# B&R Automation Studio project Nitto (part 6)

#### l2str.ab
```automation-basic
(********************************************************************
 * COPYRIGHT -- Microsoft
 ********************************************************************
 * Library: HlpStr
 * File: l2str.ab
 * Author: beutert
 * Created: March 25, 2011
 ********************************************************************
 * Implementation of library HlpStr
 ********************************************************************
 Function: convert an UDINT value to string

    input:  value (UDINT)
						pointer to string (UDINT)
   output:  strlen (UINT)
 ********************************************************************)

FUNCTION l2str
	brsstrcpy(pString,"");

	lRest = value;

	if (value > 0) then
		loop ii=9 downto 0 do
			lDivisor = UDINT(brmpow(10,ii));
			lQuot = lRest / lDivisor;
			lRest = lRest MOD lDivisor;
			if (lRest <> value) then
				brsitoa(lQuot, adr(szQuot));
				brsstrcat(pString, adr(szQuot));
			endif
		endloop;
	else
		brsstrcpy(pString,"0");
	endif;

	l2str = UINT(brsstrlen(pString));

END_FUNCTION
```

#### RTRIM.ab
```automation-basic
(********************************************************************
 * COPYRIGHT -- Microsoft
 ********************************************************************
 * Library: HlpStr
 * File: RTRIM.ab
 * Author: beutert
 * Created: April 08, 2011
 ********************************************************************
 * Implementation of library HlpStr
 ********************************************************************
 Function: delete blanks at end of string

    input:  pointer to string (UDINT)
   output:  status
 ********************************************************************)

FUNCTION RTRIM
	if (enable = true) then
		wStrLenHlp = UINT(sizeof(szHlpStr1) - 1);
		wStrLen = UINT(brsstrlen(pString));
		if (wStrLen > wStrLenHlp) then
			status = 50000;	//string too long
		else
			status = 65535;
			brsstrcpy(adr(szHlpStr1),pString);
			loop
				pByte access adr(szHlpStr1)+ wStrLen-1;
				bDbg = pByte;	//nur für Monitor
				if (pByte = ' ') then
					szHlpStr1 = LEFT(szHlpStr1, INT(wStrLen) - 1);
					wStrLen = wStrLen - 1;
				else
					exitif (1=1);
				endif;
			endloop;
			brsstrcpy(pString,adr(szHlpStr1));
			status = 0;
		endif;
	else
		status = 65534;
	endif;
	RTRIM = status;
END_FUNCTION
```

#### TRIM.ab
```automation-basic
(********************************************************************
 * COPYRIGHT -- Microsoft
 ********************************************************************
 * Library: HlpStr
 * File: TRIM.ab
 * Author: beutert
 * Created: April 08, 2011
 ********************************************************************
 * Implementation of library HlpStr
 ********************************************************************
 Function: delete blanks at beginning and end of string

    input:  pointer to string (UDINT)
   output:  status
 ********************************************************************)

FUNCTION TRIM
	if (enable = true) then
		status = RTRIM(enable, pString);
		if (status = 0) then
			status = LTRIM(enable, pString);
		endif;
	else
		status = 65534;
	endif;
	TRIM = status;
END_FUNCTION
```

### Library Logical/Libraries/SwitchConf (IEC, version 1.01.0)
Depends on: Acp10man, Acp10_MC

#### SwitchConf.typ - Exported data types
```iecst
(********************************************************************
 * COPYRIGHT -- Bernecker + Rainer
 ********************************************************************
 * Library: SwitchConf
 * File: SwitchConf.typ
 * Author: hagera
 * Created: March 01, 2010
 ********************************************************************
 * Data types of library SwitchConf
 ********************************************************************)

TYPE
	StepDescription_typ :
		( (*STEP description typ*)
		WAIT := 0, (*wait for start command*)
		CHECK_INPUT_DATA, (*check input data for FB*)
		GET_OFFSET_POS_END_SWITCH, (*get offset for positive end switch*)
		GET_OFFSET_NEG_END_SWITCH, (*get offstet for negative end switch*)
		GET_OFFSET_REF_SWITCH, (*get offset for reference switch*)
		DEFINE_PARAMETER_LIST, (*define entries for parameter list*)
		WRITE_PARAMETER_LIST (*write parameter list to axis*)
		);
	SwitchConfiguration_typ : 	STRUCT  (*single switch configuration typ*)
		ioInformation : PLACTION_GET_CROSSLINK_INFO_typ; (*i/o information for switch*)
		Status : UINT; (*status of i/o information*)
		Offset : UINT; (*offset of i/o in data*)
		shiftBits : UINT; (*bits to shift*)
	END_STRUCT;
	SwitchesACPm_typ : 	STRUCT  (*switches for ACPm typ*)
		posEndSwitch : SwitchConfiguration_typ; (*positive end switch*)
		negEndSwitch : SwitchConfiguration_typ; (*negative end switch*)
		refSwitch : SwitchConfiguration_typ; (*reference switch*)
	END_STRUCT;
	ErrorNumbers_typ :
		(
		OK := 0, (*no error*)
		INVALID_AXIS_REFERENCE := 50001, (*error number for invalid axis reference*)
		INVALID_DEVICE_NAME, (*error number for invalid device name*)
		INVALID_CHANNEL_NAME, (*error number for invalid channel name*)
		ERROR_GET_OFFSET_FOR_SWITCH, (*error number for getting offset for switch*)
		ERROR_WRITE_PARAMETER_LIST (*error number for writing parameter list*)
		);
	ParameterList_typ : 	STRUCT  (*parameter list typ*)
		List : ARRAY[0..30] OF ACP10PRB06_typ; (*parameter list*)
		listInfo : ACP10DATBL_typ; (*parameter list info*)
		configMaCyclicPos : ARRAY[0..1] OF UINT; (*MaCyclicPos*)
		ui2 : UINT; (*value data type UINT*)
		ui4 : UDINT; (*value data type UDINT*)
		Execute : BOOL; (*execute parameter list write*)
		Counter : USINT; (*parameter counter*)
	END_STRUCT;
END_TYPE
```

#### SwitchConf.fun - Exported functions and function blocks
```iecst
(********************************************************************
 * COPYRIGHT -- Bernecker + Rainer
 ********************************************************************
 * Library: SwitchConf
 * File: SwitchConf.fun
 * Author: hagera
 * Created: March 01, 2010
 ********************************************************************
 * Functions and function blocks of library SwitchConf
 ********************************************************************)

FUNCTION_BLOCK SwitchConfiguration (*FUB to configure end-switches and ref-switch for AcoposMulti*)
	VAR_INPUT
		Axis : UDINT; (*axis reference*)
		Execute : BOOL; (*start initialization at rising edge*)
		posEndSwitchDeviceName : UDINT; (*device name of module where positive end switch is connected*)
		posEndSwitchChannelName : UDINT; (*channel name of i/o where positive end switch is connected*)
		negEndSwitchDeviceName : UDINT; (*device name of module where negative end switch is connected*)
		negEndSwitchChannelName : UDINT; (*channel name of i/o where negative end switch is connected*)
		refSwitchDeviceName : UDINT; (*device name of module where reference switch is connected*)
		refSwitchChannelName : UDINT; (*channel name of i/o where reference switch is connected*)
	END_VAR
	VAR_OUTPUT
		Done : BOOL; (*initialization complete*)
		Busy : BOOL; (*initialization active*)
		Error : BOOL; (*error occured in FB*)
		ErrorID : ErrorNumbers_typ; (*error number*)
		ErrorInitparalist :UINT;
	END_VAR
	VAR
		zzEdge00000 :BOOL;
		Step : StepDescription_typ; (*intern variable*)
		Switches : SwitchesACPm_typ; (*intern variable*)
		Parameter : ParameterList_typ; (*intern variable*)
		MC_BR_InitParList_Switch : MC_BR_InitParList; (*intern variable*)
	END_VAR
END_FUNCTION_BLOCK
```

#### SwitchConfiguration.st - FUB to configure end-switches and ref-switch for ACOPOSmulti
```iecst
(********************************************************************
 * COPYRIGHT -- Bernecker + Rainer
 ********************************************************************
 * Library: SwitchConf
 * File: SwitchConfiguration.st
 * Author: hagera
 * Created: March 01, 2010
 ********************************************************************
 * Implementation of library SwitchConf
 *
 * History:
 * 2012-07-25 /schoenefeldr/
 * 		Change IPL-mode of ACP10PAR_MAx_CYCLIC_POS only if it is used
 *
 *
 *
 *
 ********************************************************************)

(* FUB to configure end-switches and ref-switch for ACOPOSmulti *)
FUNCTION_BLOCK SwitchConfiguration

CASE Step OF
	WAIT:
		IF (EDGEPOS(Execute) = 1) THEN
			Done := 0;
			Busy := 1;
			Error := 0;
			ErrorID := 0;
			Step := CHECK_INPUT_DATA;
		END_IF

	CHECK_INPUT_DATA :
		IF (Axis = 0) THEN
			Busy := 0;
			Error := 1;
			ErrorID := INVALID_AXIS_REFERENCE;
			Step := WAIT;
		ELSIF (posEndSwitchDeviceName = 0 AND negEndSwitchDeviceName = 0 AND refSwitchDeviceName = 0) OR
			(posEndSwitchDeviceName = 0 AND posEndSwitchChannelName <> 0) OR
   			(negEndSwitchDeviceName = 0 AND negEndSwitchChannelName <> 0) OR
   			(refSwitchDeviceName = 0 AND refSwitchChannelName <> 0)	THEN
			Busy := 0;
			Error := 1;
			ErrorID := INVALID_DEVICE_NAME;
			Step := WAIT;
		ELSIF (posEndSwitchDeviceName <> 0 AND posEndSwitchChannelName = 0) OR
			(negEndSwitchDeviceName <> 0 AND negEndSwitchChannelName = 0) OR
			(refSwitchDeviceName <> 0 AND refSwitchChannelName = 0) THEN
   			Busy := 0;
			Error := 1;
			ErrorID := INVALID_CHANNEL_NAME;
			Step := WAIT;
		ELSE
			Step := GET_OFFSET_POS_END_SWITCH;
		END_IF

	GET_OFFSET_POS_END_SWITCH :
		IF (posEndSwitchDeviceName = 0) THEN
			Step := GET_OFFSET_NEG_END_SWITCH;
		ELSE
			Switches.posEndSwitch.ioInformation.DeviceName := posEndSwitchDeviceName;
			Switches.posEndSwitch.ioInformation.ChannelName := posEndSwitchChannelName;

			Switches.posEndSwitch.Status := plAction(0, plACTION_GET_CROSSLINK_INFO, ADR(Switches.posEndSwitch.ioInformation), SIZEOF(Switches.posEndSwitch.ioInformation));

			IF (Switches.posEndSwitch.Status = 0) THEN
				Switches.posEndSwitch.Offset := (Switches.posEndSwitch.ioInformation.Offset / 32) * 32;
				Switches.posEndSwitch.shiftBits := Switches.posEndSwitch.ioInformation.Offset MOD 32;
				Step := GET_OFFSET_NEG_END_SWITCH;
			ELSE
				Busy := 0;
				Error := 1;
				ErrorID := ERROR_GET_OFFSET_FOR_SWITCH;
				Step := WAIT;
   			END_IF
		END_IF

	GET_OFFSET_NEG_END_SWITCH :
		IF (negEndSwitchDeviceName = 0) THEN
			Step := GET_OFFSET_REF_SWITCH;
		ELSE
			Switches.negEndSwitch.ioInformation.DeviceName := negEndSwitchDeviceName;
			Switches.negEndSwitch.ioInformation.ChannelName := negEndSwitchChannelName;

			Switches.negEndSwitch.Status := plAction(0, plACTION_GET_CROSSLINK_INFO, ADR(Switches.negEndSwitch.ioInformation), SIZEOF(Switches.negEndSwitch.ioInformation));

			IF (Switches.negEndSwitch.Status = 0) THEN
				Switches.negEndSwitch.Offset := (Switches.negEndSwitch.ioInformation.Offset / 32) * 32;
				Switches.negEndSwitch.shiftBits := Switches.negEndSwitch.ioInformation.Offset MOD 32;
				Step := GET_OFFSET_REF_SWITCH;
			ELSE
				Busy := 0;
				Error := 1;
				ErrorID := ERROR_GET_OFFSET_FOR_SWITCH;
				Step := WAIT;
   			END_IF
		END_IF

	GET_OFFSET_REF_SWITCH  :
		IF (refSwitchDeviceName = 0) THEN
			Step := DEFINE_PARAMETER_LIST;
		ELSE
			Switches.refSwitch.ioInformation.DeviceName := refSwitchDeviceName;
			Switches.refSwitch.ioInformation.ChannelName := refSwitchChannelName;

			Switches.refSwitch.Status := plAction(0, plACTION_GET_CROSSLINK_INFO, ADR(Switches.refSwitch.ioInformation), SIZEOF(Switches.refSwitch.ioInformation));

			IF (Switches.refSwitch.Status = 0) THEN
				Switches.refSwitch.Offset := (Switches.refSwitch.ioInformation.Offset / 32) * 32;
				Switches.refSwitch.shiftBits := Switches.refSwitch.ioInformation.Offset MOD 32;
				Step := DEFINE_PARAMETER_LIST;
			ELSE
				Busy := 0;
				Error := 1;
				ErrorID := ERROR_GET_OFFSET_FOR_SWITCH;
				Step := WAIT;
   			END_IF
		END_IF

	DEFINE_PARAMETER_LIST :
		Parameter.List[0].par_id := ACP10PAR_FUNCTION_BLOCK_CREATE;
		Parameter.ui2 := ACP10PAR_BIT_MODE;
		memcpy(ADR(Parameter.List[0].data_byte[0]), ADR(Parameter.ui2), SIZEOF(Parameter.ui2));
		Parameter.Counter := Parameter.Counter + 1;

		Parameter.List[Parameter.Counter].par_id := ACP10PAR_BIT_A1;
		Parameter.ui4 := 1;
		memcpy(ADR(Parameter.List[Parameter.Counter].data_byte[0]), ADR(Parameter.ui4), SIZEOF(Parameter.ui4));
		Parameter.Counter := Parameter.Counter + 1;

		Parameter.List[Parameter.Counter].par_id := ACP10PAR_BIT_A2;
		Parameter.ui4 := 1;
		memcpy(ADR(Parameter.List[Parameter.Counter].data_byte[0]), ADR(Parameter.ui4), SIZEOF(Parameter.ui4));
		Parameter.Counter := Parameter.Counter + 1;

		Parameter.List[Parameter.Counter].par_id := ACP10PAR_BIT_A3;
		Parameter.ui4 := 1;
		memcpy(ADR(Parameter.List[Parameter.Counter].data_byte[0]), ADR(Parameter.ui4), SIZEOF(Parameter.ui4));
		Parameter.Counter := Parameter.Counter + 1;

		Parameter.List[Parameter.Counter].par_id := ACP10PAR_BIT_IN1_PARID;
		Parameter.ui2 := ACP10PAR_MA1_CYCLIC_POS;
		memcpy(ADR(Parameter.List[Parameter.Counter].data_byte[0]), ADR(Parameter.ui2), SIZEOF(Parameter.ui2));
		Parameter.Counter := Parameter.Counter + 1;

		Parameter.List[Parameter.Counter].par_id := ACP10PAR_BIT_IN2_PARID;
		Parameter.ui2 := ACP10PAR_MA2_CYCLIC_POS;
		memcpy(ADR(Parameter.List[Parameter.Counter].data_byte[0]), ADR(Parameter.ui2), SIZEOF(Parameter.ui2));
		Parameter.Counter := Parameter.Counter + 1;

		Parameter.List[Parameter.Counter].par_id := ACP10PAR_BIT_IN3_PARID;
		Parameter.ui2 := ACP10PAR_MA3_CYCLIC_POS;
		memcpy(ADR(Parameter.List[Parameter.Counter].data_byte[0]), ADR(Parameter.ui2), SIZEOF(Parameter.ui2));
		Parameter.Counter := Parameter.Counter + 1;

		Parameter.List[Parameter.Counter].par_id := ACP10PAR_BIT_MODE;
		Parameter.ui2 := 10;
		memcpy(ADR(Parameter.List[Parameter.Counter].data_byte[0]), ADR(Parameter.ui2), SIZEOF(Parameter.ui2));
		Parameter.Counter := Parameter.Counter + 1;

		IF (posEndSwitchDeviceName <> 0) THEN
			// 2012-07-25 /schoenefeldr/
			// Moved here into configuration dependent section
			Parameter.List[Parameter.Counter].par_id := ACP10PAR_MA1_CYCLIC_IPL_MODE;
			Parameter.List[Parameter.Counter].data_byte[0] := 0;
			Parameter.Counter := Parameter.Counter + 1;

			Parameter.List[Parameter.Counter].par_id := ACP10PAR_CYCLIC_DP_DATA_OFFSET;
			Parameter.ui2 := Switches.posEndSwitch.Offset;
			memcpy(ADR(Parameter.List[Parameter.Counter].data_byte[0]), ADR(Parameter.ui2), SIZEOF(Parameter.ui2));
			Parameter.Counter := Parameter.Counter + 1;

			Parameter.List[Parameter.Counter].par_id := ACP10PAR_CYCLIC_DP_DATA_TYPE;
			Parameter.ui2 := 7;
			memcpy(ADR(Parameter.List[Parameter.Counter].data_byte[0]), ADR(Parameter.ui2), SIZEOF(Parameter.ui2));
			Parameter.Counter := Parameter.Counter + 1;

			Parameter.configMaCyclicPos[0] := Switches.posEndSwitch.ioInformation.NodeId;
			Parameter.configMaCyclicPos[1] := ACP10PAR_CYCLIC_DP_DATA_OFFSET;

			Parameter.List[Parameter.Counter].par_id := ACP10PAR_CONFIG_MA1_CYCLIC_POS;
			memcpy(ADR(Parameter.List[Parameter.Counter].data_byte[0]), ADR(Parameter.configMaCyclicPos), SIZEOF(Parameter.configMaCyclicPos));
			Parameter.Counter := Parameter.Counter + 1;

			Parameter.List[Parameter.Counter].par_id := ACP10PAR_BIT_B1+0;
			Parameter.ui4 := Switches.posEndSwitch.shiftBits;
			memcpy(ADR(Parameter.List[Parameter.Counter].data_byte[0]), ADR(Parameter.ui4), SIZEOF(Parameter.ui4));
			Parameter.Counter := Parameter.Counter + 1;

			Parameter.List[Parameter.Counter].par_id := ACP10PAR_POS_LIMIT_SWITCH_PARID;
			Parameter.ui2 := ACP10PAR_BIT_VALUE1;
			memcpy(ADR(Parameter.List[Parameter.Counter].data_byte[0]), ADR(Parameter.ui2), SIZEOF(Parameter.ui2));
			Parameter.Counter := Parameter.Counter + 1;
		END_IF

		IF (negEndSwitchDeviceName <> 0) THEN
			// 2012-07-25 /schoenefeldr/
			// Moved here into configuration dependent section
			Parameter.List[Parameter.Counter].par_id := ACP10PAR_MA2_CYCLIC_IPL_MODE;
			Parameter.List[Parameter.Counter].data_byte[0] := 0;
			Parameter.Counter := Parameter.Counter + 1;

			Parameter.List[Parameter.Counter].par_id := ACP10PAR_CYCLIC_DP_DATA_OFFSET;
			Parameter.ui2 := Switches.negEndSwitch.Offset;
			memcpy(ADR(Parameter.List[Parameter.Counter].data_byte[0]), ADR(Parameter.ui2), SIZEOF(Parameter.ui2));
			Parameter.Counter := Parameter.Counter + 1;

			Parameter.List[Parameter.Counter].par_id := ACP10PAR_CYCLIC_DP_DATA_TYPE;
			Parameter.ui2 := 7;
			memcpy(ADR(Parameter.List[Parameter.Counter].data_byte[0]), ADR(Parameter.ui2), SIZEOF(Parameter.ui2));
			Parameter.Counter := Parameter.Counter + 1;

			Parameter.configMaCyclicPos[0] := Switches.negEndSwitch.ioInformation.NodeId;
			Parameter.configMaCyclicPos[1] := ACP10PAR_CYCLIC_DP_DATA_OFFSET;

			Parameter.List[Parameter.Counter].par_id := ACP10PAR_CONFIG_MA2_CYCLIC_POS;
			memcpy(ADR(Parameter.List[Parameter.Counter].data_byte[0]), ADR(Parameter.configMaCyclicPos), SIZEOF(Parameter.configMaCyclicPos));
			Parameter.Counter := Parameter.Counter + 1;

			Parameter.List[Parameter.Counter].par_id := ACP10PAR_BIT_B2+0;
			Parameter.ui4 := Switches.negEndSwitch.shiftBits;
			memcpy(ADR(Parameter.List[Parameter.Counter].data_byte[0]), ADR(Parameter.ui4), SIZEOF(Parameter.ui4));
			Parameter.Counter := Parameter.Counter + 1;

			Parameter.List[Parameter.Counter].par_id := ACP10PAR_NEG_LIMIT_SWITCH_PARID;
			Parameter.ui2 := ACP10PAR_BIT_VALUE2;
			memcpy(ADR(Parameter.List[Parameter.Counter].data_byte[0]), ADR(Parameter.ui2), SIZEOF(Parameter.ui2));
			Parameter.Counter := Parameter.Counter + 1;
		END_IF

		IF (refSwitchDeviceName <> 0) THEN
			// 2012-07-25 /schoenefeldr/
			// Moved here into configuration dependent section
			Parameter.List[Parameter.Counter].par_id := ACP10PAR_MA3_CYCLIC_IPL_MODE;
			Parameter.List[Parameter.Counter].data_byte[0] := 0;
			Parameter.Counter := Parameter.Counter + 1;

			Parameter.List[Parameter.Counter].par_id := ACP10PAR_CYCLIC_DP_DATA_OFFSET;
			Parameter.ui2 := Switches.refSwitch.Offset;
			memcpy(ADR(Parameter.List[Parameter.Counter].data_byte[0]), ADR(Parameter.ui2), SIZEOF(Parameter.ui2));
			Parameter.Counter := Parameter.Counter + 1;

			Parameter.List[Parameter.Counter].par_id := ACP10PAR_CYCLIC_DP_DATA_TYPE;
			Parameter.ui2 := 7;
			memcpy(ADR(Parameter.List[Parameter.Counter].data_byte[0]), ADR(Parameter.ui2), SIZEOF(Parameter.ui2));
			Parameter.Counter := Parameter.Counter + 1;

			Parameter.configMaCyclicPos[0] := Switches.refSwitch.ioInformation.NodeId;
			Parameter.configMaCyclicPos[1] := ACP10PAR_CYCLIC_DP_DATA_OFFSET;

			Parameter.List[Parameter.Counter].par_id := ACP10PAR_CONFIG_MA3_CYCLIC_POS;
			memcpy(ADR(Parameter.List[Parameter.Counter].data_byte[0]), ADR(Parameter.configMaCyclicPos), SIZEOF(Parameter.configMaCyclicPos));
			Parameter.Counter := Parameter.Counter + 1;

			Parameter.List[Parameter.Counter].par_id := ACP10PAR_BIT_B3+0;
			Parameter.ui4 := Switches.refSwitch.shiftBits;
			memcpy(ADR(Parameter.List[Parameter.Counter].data_byte[0]), ADR(Parameter.ui4), SIZEOF(Parameter.ui4));
			Parameter.Counter := Parameter.Counter + 1;

			Parameter.List[Parameter.Counter].par_id := ACP10PAR_REFERENCE_SWITCH_PARID;
			Parameter.ui2 := ACP10PAR_BIT_VALUE3;
			memcpy(ADR(Parameter.List[Parameter.Counter].data_byte[0]), ADR(Parameter.ui2), SIZEOF(Parameter.ui2));
			Parameter.Counter := Parameter.Counter + 1;
		END_IF

		Step := WRITE_PARAMETER_LIST;

	WRITE_PARAMETER_LIST :
		Parameter.listInfo.parameter.data_adr := ADR(Parameter.List);
		Parameter.listInfo.parameter.format := ncFORMAT_B06;
		Parameter.listInfo.parameter.data_len := Parameter.Counter * SIZEOF(ACP10PRB06_typ);
		Parameter.Execute := 1;

		IF (MC_BR_InitParList_Switch.Done = 1) THEN
			Parameter.Execute := 0;
			Busy := 0;
			Done := 1;
			Step := WAIT;
		ELSIF (MC_BR_InitParList_Switch.Error = 1) THEN
			Parameter.Execute := 0;
			Busy := 0;
			ErrorInitparalist := MC_BR_InitParList_Switch.ErrorID;
			Error := 1;
			ErrorID := ERROR_WRITE_PARAMETER_LIST;
			Step := WAIT;
		END_IF

		MC_BR_InitParList_Switch(Axis := Axis, Execute := Parameter.Execute, DataAddress := ADR(Parameter.listInfo));

END_CASE

END_FUNCTION_BLOCK
```

### Library Logical/Libraries/TorqueCtrl (IEC) - Torque control
Depends on: LoopConR, Acp10_MC

#### TorqueCtrl.typ - Exported data types
```iecst
(********************************************************************
 * COPYRIGHT -- Bernecker + Rainer
 ********************************************************************
 * Library: TorqueCtrl
 * File: TorqueCtrl.typ
 * Author: knausenbergl
 * Created: October 29, 2012
 ********************************************************************
 * Data types of library TorqueCtrl
 ********************************************************************)

TYPE
	TC_WINDER_IS_TYP : 	STRUCT
		RefTension : ARRAY[0..1]OF REAL;
		RefDiameter : ARRAY[0..1]OF REAL;
		SetLineSpeed : REAL;
		ActDiameter : REAL;
		SetWndSpeed : REAL;
		SetMotorTorque : REAL;
		LineUnits : REAL;
		LCRLimScal_Tension : LCRLimScal; (*scale tension force depending on actual diameter*)
		GearRatio : REAL;
		EncoderIf : ACP10ENCPA_typ;
		WndUnitsPerLoadRev : REAL; (*winder units per load revolution [Slave Units]*)
		SetTorqueRaw : REAL; (*raw, unlimited set torque [Nm]*)
		SetTension : REAL;
	END_STRUCT;
END_TYPE
```

#### TorqueCtrl.fun - Exported functions and function blocks
```iecst
(********************************************************************
 * COPYRIGHT -- Bernecker + Rainer
 ********************************************************************
 * Library: TorqueCtrl
 * File: TorqueCtrl.fun
 * Author: knausenbergl
 * Created: October 29, 2012
 ********************************************************************
 * Functions and function blocks of library TorqueCtrl
 ********************************************************************)

FUNCTION_BLOCK TC_Winder
	VAR_INPUT
		RefTension : ARRAY[0..1] OF REAL; (*reference material tension [N]*)
		RefDiameter : ARRAY[0..1] OF REAL; (*reference diameters corresponding to RefTension [Master Units]*)
		SetLineSpeed : REAL; (*line speed [Master Units / s]*)
		ActDiameter : REAL; (*actual winder diameter [Master Units]*)
		EncoderIf : ACP10ENCPA_typ; (*winder encoder interface*)
		GearRatio : REAL; (*motor rev. / winder rev. []*)
		LineUnits : REAL; (*line position scaling [Master Units / m]*)
	END_VAR
	VAR_OUTPUT
		SetWndSpeed : REAL; (*set winder speed [Slave Units / s]*)
		SetMotorTorque : REAL; (*set motor torque [Nm]*)
		SetTension : REAL; (*set material tension [N]*)
	END_VAR
	VAR
		IS : TC_WINDER_IS_TYP; (*internal data*)
	END_VAR
END_FUNCTION_BLOCK
```

#### TC_Winder.st
```iecst
(********************************************************************
 * COPYRIGHT -- Bernecker + Rainer
 ********************************************************************
 * Library: TorqueCtrl
 * File: TC_Winder.st
 * Author: knausenbergl
 * Created: October 29, 2012
 ********************************************************************
 * Implementation of library TorqueCtrl
 *
 * History:
 * 2012-10-29 /knausenbergl/
 *		Task created
 * 2012-10-31 /schoenefeldr/
 *		Removed unused dynamic adaptation of force
 * 2012-11-01 /schoenefeldr/
 *		Removed unused inputs
 ********************************************************************)

(* Calculate velocity and torque depending on force setpoint and diameter *)
FUNCTION_BLOCK TC_Winder

	//UPDATE FUB INPUTS
	IS.RefTension		:= RefTension;
	IS.RefDiameter		:= RefDiameter;
	IS.SetLineSpeed		:= SetLineSpeed;
	IS.ActDiameter		:= ActDiameter;
	IS.EncoderIf		:= EncoderIf;
	IS.GearRatio		:= GearRatio;
	IS.LineUnits		:= LineUnits;

	IS.WndUnitsPerLoadRev	:= UDINT_TO_REAL(IS.EncoderIf.scaling.load.units) * IS.GearRatio / UDINT_TO_REAL(IS.EncoderIf.scaling.load.rev_motor);

	//calculate set winder speed
	IF (IS.ActDiameter > 0.0) THEN
		IS.SetWndSpeed	:= IS.SetLineSpeed / (MATH_PI * IS.ActDiameter) * IS.WndUnitsPerLoadRev;
	ELSE
		IS.SetWndSpeed	:= 0.0;
	END_IF;

	//calculate set tension depending on actual diameter
	IS.LCRLimScal_Tension.x		:= IS.ActDiameter;
	IS.LCRLimScal_Tension.x1	:= IS.RefDiameter[0];
	IS.LCRLimScal_Tension.y1	:= IS.RefTension[0];
	IS.LCRLimScal_Tension.x2	:= IS.RefDiameter[1];
	IS.LCRLimScal_Tension.y2	:= IS.RefTension[1];
	IS.LCRLimScal_Tension();
	IS.SetTension	:= IS.LCRLimScal_Tension.y;
	IS.SetTorqueRaw	:= IS.LCRLimScal_Tension.y * IS.ActDiameter / (2.0 * IS.GearRatio * IS.LineUnits);

	//UPDATE FUB OUTPUTS
	SetWndSpeed		:= IS.SetWndSpeed;
	SetMotorTorque	:= IS.SetTorqueRaw;
	SetTension		:= IS.SetTension;

END_FUNCTION_BLOCK
```

### Library Logical/Libraries/UserVC (IEC, version 3.00.0)
Depends on: AsString, runtime

#### UserVC.var
```iecst
VAR CONSTANT
	ENABLE_NOT_SET	:UINT	:=65000;
	HEX_BASE	:SINT	:=16;
	SORTING_ABORTED	:UINT	:=6000;
	SORTING_BUSY	:UINT	:=65535;
	SORTING_NO_ERROR	:UINT	:=0;
	SORT_ALPHANUMERICALLY	:USINT	:=4;
	SORT_CASE_SENSITIVE1	:USINT	:=2;
	SORT_CASE_SENSITIVE2	:USINT	:=3;
	SWAP_FILENAMES	:USINT	:=1;
END_VAR
```

#### UserVC.fun
```iecst
FUNCTION_BLOCK Sort
	VAR_INPUT
		enable : BOOL;
		pStringArray : UDINT;
		StringLen : UINT;
		ArrayLen : UINT;
	END_VAR
	VAR_OUTPUT
		Status : UINT;
	END_VAR
	VAR
		xcnt : UINT;
		ycnt : UINT;
		StepCounter : UINT;
		SortStep : USINT;
		FileNameBuffer : STRING[80];
		pChar1 : REFERENCE TO USINT;
		pChar2 : REFERENCE TO USINT;
	END_VAR
END_FUNCTION_BLOCK

FUNCTION_BLOCK ConvertHex
	VAR_INPUT
		Enable : BOOL;
		pHexValue : UDINT;
		DecValue : UDINT;
		SizeDecValue : USINT;
	END_VAR
	VAR_OUTPUT
		Status : UINT;
	END_VAR
	VAR
		HexASCII : ARRAY[0..7] OF USINT;
		Index : SINT;
		End : USINT;
		Rest : UDINT;
	END_VAR
END_FUNCTION_BLOCK
```

#### Sort.st
```iecst
FUNCTION_BLOCK Sort
(* Implementation of sort *)

(**********************************************************************************************************************)
(* Object name: sort                                                                                                                              	*)
(* Author:      Peter Hauser,  B&R                                                                                                               	*)
(* Site:        Eggelsberg                                                                                                                             	*)
(* Created:     25-aug-2003                                                                                                                           	*)
(* Restriction: ------                                                                                                                          	*)
(* Description: The Sort-Function sorts a String Array alphanumerically                                                                                                                                       	*)
(*                                                                                                                                                              	*)
(*----------------------------------------------------------------------------------------------------------------------------------------	*)
(* Version 1.00.1   25-aug-2003  Peter Hauser									*)
(*----------------------------------------------------------------------------------------------------------------------------------------	*)
(* Development tool: B&R Automation Studio V2.3.0.9 							*)
(*----------------------------------------------------------------------------------------------------------------------------------------	*)
(* Comment:                                                                                                                     			*)
(**********************************************************************************************************************)

(* Errors *)

IF ((enable = 0) AND (StepCounter > 0) AND (StepCounter < ((ArrayLen / StringLen) - 1))) THEN
	Status:= SORTING_ABORTED;

ELSIF ((enable = 1) AND (StepCounter >= 0) AND (StepCounter < ((ArrayLen / StringLen) - 1))) THEN
	Status:= SORTING_BUSY;

ELSE
	Status:= SORTING_NO_ERROR;

END_IF

(* sorting StringArray alphanumerically *)

IF ((enable = 1) AND ((Status = 0) OR (Status = 65535))) THEN

	FOR xcnt:= 0 TO ((ArrayLen / StringLen) - 2) DO

		FOR ycnt:= 0 TO StringLen DO
			(* read characters of FileNames *)
			pChar1 ACCESS (pStringArray + (StringLen * xcnt) + ycnt);
			pChar2 ACCESS (pStringArray + (StringLen * xcnt) + StringLen + ycnt);

			(* if no data in FileName1 -> Swap FileNames *)
			IF ((ycnt = 0) AND (pChar1 = 0) AND (pChar2 > 0)) THEN
				SortStep:= SWAP_FILENAMES;

			(* if no data in FileName2 -> next 2 FileNames *)
			ELSIF ((ycnt = 0) AND (pChar2 = 0)) THEN
				EXIT;

			(* if data in both FileNames *)
			ELSE
				(* detect case of letters *)
				IF ((pChar1 >= 65) AND (pChar1 <= 90) AND (pChar2 >= 97) AND (pChar2 <= 122)) THEN
					SortStep:= SORT_CASE_SENSITIVE1;

				ELSIF ((pChar1 >= 97) AND (pChar1 <= 122) AND (pChar2 >= 65) AND (pChar2 <= 90)) THEN
					SortStep:= SORT_CASE_SENSITIVE2;

				(* if characters are equal -> compare next characters of FileName *)
				ELSIF ((pChar1 = pChar2) AND (pChar2 <> 0)) THEN
					SortStep:= 0;

				(* if both FileNames are finished *)
				ELSIF ((pChar1 = 0) AND (pChar2 = 0)) THEN
					EXIT;

				(* sort Alphanumerically *)
				ELSE
					SortStep:= SORT_ALPHANUMERICALLY;
				END_IF
			END_IF

			CASE SortStep OF

				SWAP_FILENAMES:
					memcpy(ADR(FileNameBuffer), (pStringArray + (StringLen * xcnt)), StringLen);
					memcpy((pStringArray + (StringLen * xcnt)), (pStringArray + (StringLen * xcnt) + StringLen), StringLen);
					memcpy((pStringArray + (StringLen * xcnt) + StringLen), ADR(FileNameBuffer), StringLen);
					EXIT;

				SORT_CASE_SENSITIVE1:
					IF (pChar2 <= (pChar1 + 32)) THEN
						memcpy(ADR(FileNameBuffer), (pStringArray + (StringLen * xcnt)), StringLen);
						memcpy((pStringArray + (StringLen * xcnt)), (pStringArray + (StringLen * xcnt) + StringLen), StringLen);
						memcpy((pStringArray + (StringLen * xcnt) + StringLen), ADR(FileNameBuffer), StringLen);
						EXIT;
					ELSE
						EXIT;
					END_IF

				SORT_CASE_SENSITIVE2:
					IF (pChar2 < (pChar1 - 32)) THEN
						memcpy(ADR(FileNameBuffer), (pStringArray + (StringLen * xcnt)), StringLen);
						memcpy((pStringArray + (StringLen * xcnt)), (pStringArray + (StringLen * xcnt) + StringLen), StringLen);
						memcpy((pStringArray + (StringLen * xcnt) + StringLen), ADR(FileNameBuffer), StringLen);
						EXIT;
					ELSE
						EXIT;
					END_IF

				SORT_ALPHANUMERICALLY:
					IF pChar1 > pChar2 THEN
						memcpy(ADR(FileNameBuffer), (pStringArray + (StringLen * xcnt)), StringLen);
						memcpy((pStringArray + (StringLen * xcnt)), (pStringArray + (StringLen * xcnt) + StringLen), StringLen);
						memcpy((pStringArray + (StringLen * xcnt) + StringLen), ADR(FileNameBuffer), StringLen);
						EXIT;
					ELSE
						EXIT;
					END_IF

			END_CASE
		END_FOR

	END_FOR

	(* execute sorting [NumStringsToSort] times *)
	IF xcnt = ((ArrayLen / StringLen) - 1) THEN
		StepCounter:= StepCounter + 1;
	END_IF;

	IF StepCounter >= (ArrayLen / StringLen) THEN
		StepCounter:= 0;
	END_IF

END_IF			(* if enable = 1 *)

END_FUNCTION_BLOCK
```

#### ConvertHex.st
```iecst
FUNCTION_BLOCK ConvertHex
(* Implementation of ConvertHex *)

(**********************************************************************************************************************)
(* Object name: ConvertHex                                                                                                                              	*)
(* Author:      Christoph Trappl,  B&R                                                                                                               	*)
(* Site:        Eggelsberg                                                                                                                             	*)
(* Created:     27-aug-2003                                                                                                                           	*)
(* Restriction: -----                                                                                                                          	*)
(* Description: Converts a decimal value to hexadecimal ASCII                                                                                                                                	*)
(*                                                                                                                                                              	*)
(*----------------------------------------------------------------------------------------------------------------------------------------	*)
(* Version 1.00.1   27-aug-2003  Christoph Trappl								*)
(*----------------------------------------------------------------------------------------------------------------------------------------	*)
(* Version 1.00.2   02-feb-2004  Peter Hauser									*)
(*----------------------------------------------------------------------------------------------------------------------------------------	*)
(* Development tool: B&R Automation Studio V2.3.0.9 							*)
(*----------------------------------------------------------------------------------------------------------------------------------------	*)
(* Comment:                                                                                                                     			*)
(**********************************************************************************************************************)

(* Execute Functionblock when enable = true *)
IF (Enable = 1) THEN

//210812,TB: CONSTANT EXECUTION_BUSY replaced	by standard
//	Status := EXECUTION_BUSY;
	Status := ERR_FUB_BUSY;

	(* reset the complete memory area, that will be overwritten during the function execution *)
	memset(pHexValue, 0, SIZEOF(HexASCII));

	HexASCII[0]:= 0;
	HexASCII[1]:= 0;
	HexASCII[2]:= 0;
	HexASCII[3]:= 0;
	HexASCII[4]:= 0;
	HexASCII[5]:= 0;
	HexASCII[6]:= 0;
	HexASCII[7]:= 0;

	IF SizeDecValue = 0 THEN
		IF (DecValue > 16#FFFFFFF)  THEN
			Index:= 7;
		ELSIF (DecValue > 16#FFFFFF) THEN
			Index:= 6;
		ELSIF (DecValue > 16#FFFFF) THEN
			Index:= 5;
		ELSIF (DecValue > 16#FFFF) THEN
			Index:= 4;
		ELSIF (DecValue > 16#FFF) THEN
			Index:= 3;
		ELSIF (DecValue > 16#FF) THEN
			Index:= 2;
		ELSIF (DecValue > 16#F) THEN
			Index:= 1;
		ELSE
			Index:= 0;
		END_IF
	ELSIF SizeDecValue = 1 THEN
		Index:= 1;
	ELSIF SizeDecValue = 2 THEN
		Index:= 3;
	ELSIF SizeDecValue = 4 THEN
		Index:= 7;
	END_IF

	REPEAT
		IF DecValue > 0 OR SizeDecValue > 0 THEN
			End:= 0;
			Rest:= DecValue MOD HEX_BASE;
			DecValue:= DecValue / HEX_BASE;

			IF ( (Rest >= 0) AND (Rest <= 9) ) THEN
				HexASCII[Index]:= UDINT_TO_USINT((48 + Rest));
			ELSE
				HexASCII[Index]:= UDINT_TO_USINT((55 + Rest));
			END_IF

			Index:= Index - 1;
		END_IF

		IF (DecValue = 0 AND SizeDecValue = 0) OR Index < 0 THEN
			Index:= 0;
			End:= 1;
		END_IF
	UNTIL
		End = 1
	END_REPEAT;

	memcpy(pHexValue, ADR(HexASCII), SIZEOF(HexASCII));
//210812,TB: CONSTANT EXECUTION_OK replaced	by standard
//	Status := EXECUTION_OK;
	Status := ERR_OK;
ELSE
	Status:= ENABLE_NOT_SET;
END_IF

END_FUNCTION_BLOCK
```

### Library Logical/Libraries/UtilTyp (IEC) - Utilities and data types

#### UtilTyp.typ - Exported data types
```iecst
(********************************************************************
 * COPYRIGHT -- Bernecker + Rainer
 ********************************************************************
 * Library: UtilTyp
 * File: UtilTyp.typ
 * Author: schoenefeldr
 * Created: July 09, 2012
 ********************************************************************
 * Data types of library UtilTyp
 ********************************************************************)
(*Digital input and output data type*)

TYPE
	DiDo_Type : 	STRUCT
		Config : DiDoCfg_Type; (*Analogue IO configuration*)
		Value : DiDoValue_Type;
	END_STRUCT;
	DiDoValue_Type : 	STRUCT
		InVal : BOOL;
		ActOut : BOOL;
		IsBlinking : BOOL;
		State : BOOL;
	END_STRUCT;
	DiDoCfg_Type : 	STRUCT  (*Contains configuration data*)
		OptionPLC : UDINT; (*Options for PLC *)
	END_STRUCT;
END_TYPE

(*Analogue input and output data type*)

TYPE
	AiAo_Type : 	STRUCT  (*Universal analogue IO data type*)
		Config : AiAoCfg_Type; (*Analogue IO configuration*)
		Value : AiAoValue_Type; (*IO values*)
	END_STRUCT;
	AiAoCfg_Type : 	STRUCT  (*Contains configuration data*)
		OptionPLC : UDINT; (*Options for PLC *)
		OptionVisu : UDINT; (*Options for visu configuration*)
		RawMax : REAL; (*Maximum of raw value*)
		RawMin : REAL; (*Minimum of raw value*)
		ScaleGain : REAL; (*Gain for scaling*)
		ScaleOffset : REAL; (*Zero offset for scaling in application units*)
	END_STRUCT;
	AiAoValue_Type : 	STRUCT  (*Contains IO values*)
		RawInt : INT; (*Raw input or output value 16 Bit*)
		RawDInt : DINT; (*Raw input or output value 32 Bit*)
		Scaled : REAL; (*Scaled physical value*)
	END_STRUCT;
END_TYPE
```

#### UtilTyp.var - Exported constants
```iecst
(********************************************************************
 * COPYRIGHT -- Bernecker + Rainer
 ********************************************************************
 * Library: UtilTyp
 * File: UtilTyp.var
 * Author: schoenefeldr
 * Created: July 09, 2012
 ********************************************************************
 * Constants of library UtilTyp
 ********************************************************************)
(*Global constants*)
VAR CONSTANT
	MATH_PI : REAL := 3.141593; (*Constant value PI*)
END_VAR
(*Definitions for configuration constants*)
VAR CONSTANT
	CONTACT_IS_OPENER : USINT := 0; (*Opener contact at input*)
END_VAR
(*Return codes*)
VAR CONSTANT
	ERR_OK : UINT := 0; (*No error*)
	ERR_DIVISION_BY_ZERO : UINT := 65534; (*Division by zero*)
	ERR_INT_OVERFLOW : UINT := 65533; (*Integer overflow, value higher than positive integer range*)
	ERR_INT_UNDERFLOW : UINT := 65532; (*Integer underflow, value lower than negaitive integer range or < 0*)
END_VAR
```

#### UtilTyp.fun - Exported functions and function blocks
```iecst
(********************************************************************
 * COPYRIGHT -- Bernecker + Rainer
 ********************************************************************
 * Library: UtilTyp
 * File: UtilTyp.fun
 * Author: schoenefeldr
 * Created: July 09, 2012
 ********************************************************************
 * Functions and function blocks of library UtilTyp
 ********************************************************************)

FUNCTION UtilScaleAin32 : UINT (*Scale analogue input 32 Bit*)
	VAR_INPUT
		dataAdr : REFERENCE TO AiAo_Type;
	END_VAR
END_FUNCTION

FUNCTION UtilScaleAin16 : UINT (*Scale analogue input 16 Bit*)
	VAR_INPUT
		dataAdr : REFERENCE TO AiAo_Type;
	END_VAR
END_FUNCTION

FUNCTION UtilScaleAout16 : UINT (*Scale a real vaue into a 16 Bit analogue output*)
	VAR_INPUT
		dataAdr : REFERENCE TO AiAo_Type;
	END_VAR
	VAR
		outValue : REAL; (*Internal limited value*)
	END_VAR
END_FUNCTION

FUNCTION_BLOCK UtilFreqPulse (*FB generates a pulse at a defined frequency*)
	VAR_INPUT
		Frequency : UDINT; (*Pulse frequency [0.1 Hz]*)
		dataAdr : REFERENCE TO DiDo_Type;
	END_VAR
	VAR
		RTInfo_0 : RTInfo;
		periodCntMax : UDINT; (*Maximum counter value for one pulse period in cycletime*)
		periodCntAct : UDINT; (*Counter for pulse period in cycletime*)
		cycletimeValue : UDINT; (*Cycletime in ms*)
		cycletimeValid : BOOL; (*internal cycletime has been determined*)
	END_VAR
END_FUNCTION_BLOCK

FUNCTION UtilGetDiameter : REAL (*Calculates a diameter from a scaled sensor value [mm] and an calibrated offset [mm]*)
	VAR_INPUT
		adr_Ain : REFERENCE TO AiAo_Type; (*address of analogue input structure*)
		offset : REAL; (*calibrated diameter offset in [mm]*)
		coreDiam : REAL; (*additional offset through core diameter in [mm]*)
	END_VAR
END_FUNCTION

FUNCTION UtilCalcSetVeloHz : REAL (*Calculate velocity setpoint in user units [0.001 Hz] from input velocity in user units [µm/s]*)
	VAR_INPUT
		FIXED_DIAM : REAL; (*Used diameter if diameter input is zero*)
		veloM : REAL; (*Velocitiy in user unit [µm/s] (direct input)*)
		diam_mm : REAL; (*diameter of winder in [mm] (assume miminum diameter if zero)*)
	END_VAR
END_FUNCTION

FUNCTION UtilGetVeloHz : REAL (*Calculate velocity in user units [0.001 Hz] from input velocity in user units [µm/s]*)
	VAR_INPUT
		veloM : REAL; (*Velocitiy in user unit [µm/s] (direct input)*)
		diam_mm : REAL; (*diameter of winder in [mm]*)
	END_VAR
END_FUNCTION

FUNCTION UtilScal : REAL (*Scaling an input via a line equation*)
	VAR_INPUT
		In : REAL; (*Input value*)
		Gain : REAL; (*line equation gain*)
		Offset : REAL; (*line equation offset*)
	END_VAR
END_FUNCTION
```

#### UtilScaleAin32.st - Scale analogue input 32 Bit
```iecst
(********************************************************************
 * COPYRIGHT -- Bernecker + Rainer
 ********************************************************************
 * Library: UtilTyp
 * File: UtilScaleAin32.st
 * Author: schoenefeldr
 * Created: July 16, 2012
 ********************************************************************
 * Implementation of library UtilTyp
 ********************************************************************)

(* Scale analogue input 32 Bit *)
FUNCTION UtilScaleAin32
	// Result is the sum of the scaled raw value (signed 32 bit) and the offset (in application units)
	dataAdr.Value.Scaled := dataAdr.Config.ScaleOffset +
							(dataAdr.Config.ScaleGain * DINT_TO_REAL( dataAdr.Value.RawDInt ));
	UtilScaleAin32 := ERR_OK;   // Return value = OK
END_FUNCTION
```

#### UtilScaleAin16.st - Scale analogue input 16 Bit
```iecst
(********************************************************************
 * COPYRIGHT -- Bernecker + Rainer
 ********************************************************************
 * Library: UtilTyp
 * File: UtilScaleAin16.st
 * Author: schoenefeldr
 * Created: July 16, 2012
 ********************************************************************
 * Implementation of library UtilTyp
 ********************************************************************)

(* Scale analogue input 16 Bit *)
FUNCTION UtilScaleAin16
	// Result is the sum of the scaled raw value (signed 16 bit) and the offset (in application units)
	dataAdr.Value.Scaled := dataAdr.Config.ScaleOffset +
							(dataAdr.Config.ScaleGain * INT_TO_REAL( dataAdr.Value.RawInt ));
	UtilScaleAin16 := ERR_OK;   // Return value = OK
END_FUNCTION
```

#### UtilScaleAout16.st - Scale a real vaue into a 16 Bit analogue output
```iecst
(********************************************************************
 * COPYRIGHT -- Bernecker + Rainer
 ********************************************************************
 * Library: UtilTyp
 * File: UtilScaleAout16.st
 * Author: schoenefeldr
 * Created: July 17, 2012
 ********************************************************************
 * Implementation of library UtilTyp
 ********************************************************************)

(* Scale a real vaue into a 16 Bit analogue output *)
FUNCTION UtilScaleAout16
	// Input is the data value that first has to be limited to the scaled range
	// (application units) and then into the limitations of the raw range
	// depending on the analogue outputs.
	outValue := dataAdr.Value.Scaled + dataAdr.Config.ScaleOffset;

	// Now scale the output value in application units into raw range
	IF NOT (dataAdr.Config.ScaleGain = 0.0) THEN
		outValue := outValue / dataAdr.Config.ScaleGain;
		UtilScaleAout16 := ERR_OK;
	ELSE
		// Invalid Scale Gain (division by zero), add offset only, no further scaling
		outValue 		:= 0.0;
		UtilScaleAout16 := ERR_DIVISION_BY_ZERO;
	END_IF

	// Limit the result to the physical limits of the analogue output
	IF outValue > dataAdr.Config.RawMax THEN
		outValue := dataAdr.Config.RawMax;
		// Second limitation to physical limit of output / conversion
		IF outValue > 32767.0 THEN
			outValue 		:= 32767.0;
			UtilScaleAout16 := ERR_INT_OVERFLOW;
		END_IF
	ELSIF outValue < dataAdr.Config.RawMin THEN
		outValue := dataAdr.Config.RawMin;
		// Second limitation to physical limit of output / conversion
		IF outValue < -32768.0 THEN
			outValue 		:= -32768.0;
			UtilScaleAout16 := ERR_INT_UNDERFLOW;
		END_IF
	END_IF
	// convert value into output
	dataAdr.Value.RawInt := REAL_TO_INT (outValue);
END_FUNCTION
```

#### UtilFreqPulse.st - FB generates a pulse at a defined frequency
```iecst
(********************************************************************
 * COPYRIGHT -- Bernecker + Rainer
 ********************************************************************
 * Library: UtilTyp
 * File: UtilFreqPulse.st
 * Author: schoenefeldr
 * Created: July 17, 2012
 ********************************************************************
 * Implementation of library UtilTyp
 *
 * History:
 * 2012-07-17 /schoenefeldr/
 *		Task created
 * 2012-10-15 /schoenefeldr/
 *		Increased internal resolution to 0.1 ms
 ********************************************************************)

(* FB generates a pulse at a defined frequency *)
FUNCTION_BLOCK UtilFreqPulse

	// Exit if frequency is 0 or no pulse requested
	IF (Frequency = 0) OR NOT dataAdr.Value.IsBlinking THEN
		dataAdr.Value.ActOut 	:= dataAdr.Value.State;
		periodCntAct			:= 0;
		RETURN;
	END_IF

	// Calculate the cycletime if necessary
	IF (NOT cycletimeValid AND dataAdr.Value.IsBlinking) THEN
 		// Call FB to determine the task cycletime
		RTInfo_0(enable := TRUE);

		// The FB returns the cycletime in µs -> convert to ms
		IF(RTInfo_0.status = 0)THEN
			// 2012-10-15 /schoenefeldr/: Increase resolution to 0.1 ms
			cycletimeValue := RTInfo_0.cycle_time / 100;
			cycletimeValid := TRUE;
		END_IF
	END_IF

	// Calculate state and derive output only if...
	// -> the data state is TRUE (output may be set)
	// -> blinking is requested
	IF (cycletimeValid AND dataAdr.Value.IsBlinking AND dataAdr.Value.State) THEN

		// Calculate period counter
		// 2012-10-15 /schoenefeldr/: Increase resolution to 0.1 ms
		periodCntMax := 100000 / Frequency;

		// The period always starts with a set output
		IF (periodCntAct > periodCntMax) THEN
			// Reset output and counter
			dataAdr.Value.ActOut 	:= FALSE;
			periodCntAct			:= 0;
		ELSIF (periodCntAct > (periodCntMax / 2)) THEN
			dataAdr.Value.ActOut 	:= FALSE;
			periodCntAct := periodCntAct + cycletimeValue;
		ELSE
			dataAdr.Value.ActOut := TRUE;
			periodCntAct := periodCntAct + cycletimeValue;
		END_IF

	ELSE
		// Reset cycle time valid flag => a valid cycletime will always be calculated
		cycletimeValid := FALSE;

	END_IF

END_FUNCTION_BLOCK
```

#### UtilGetDiameter.st - Calculates a diameter from a scaled sensor value [mm] and an calibrated offset [mm]
```iecst
(********************************************************************
 * COPYRIGHT -- Bernecker + Rainer
 ********************************************************************
 * Library: UtilTyp
 * File: UtilGetDiameter.st
 * Author: schoenefeldr
 * Created: August 01, 2012
 *
 *
 * History:
 * 2012-09-20 /schoenefeldr/
 * 		core diameter as additional input
 *
 ********************************************************************
 * Implementation of library UtilTyp
 ********************************************************************)

(* Calculates a diameter from a scaled sensor value [mm] and an calibrated offset [mm] *)
FUNCTION UtilGetDiameter
	// This function calculates the diameter from a distance value as input [mm]
	// and an offset derived from the distance value for an "empty" winder.
	UtilGetDiameter	:= ((offset + (coreDiam / 2.0)) - adr_Ain.Value.Scaled) * 2;
	IF UtilGetDiameter < 0.0 THEN
		// Invalid diameter, return 0.0
		UtilGetDiameter := 0.0;
	END_IF
END_FUNCTION
```

#### UtilCalcSetVeloHz.st - Calculate velocity setpoint in user units [0.001 Hz] from input velocity in user units [µm/s]
```iecst
(********************************************************************
 * COPYRIGHT -- Bernecker + Rainer
 ********************************************************************
 * Library: UtilTyp
 * File: UtilCalcSetVeloHz.st
 * Author: schoenefeldr
 * Created: August 02, 2012
 ********************************************************************
 * Implementation of library UtilTyp
 ********************************************************************)

(* Calculate velocity setpoint in user units [0.001 Hz] from input velocity in user units [µm/s] *)
FUNCTION UtilCalcSetVeloHz
	// Formula:
	// 					n [0.001 Hz] = ( v [m/s] / (pi * diam [m]) ) * 1.000
	// normalized		n [0.001 Hz] = ( ( v [µm/s] / 1.000.000 ) / (pi * ( diam [mm] / 1.000 ) ) ) * 1.000
	// reduced:			n [0.001 Hz] = ( ( v [µm/s] / 1.000 ) / (pi * ( diam [mm] / 1.000 ) ) ) * 1
	// finally reduced:	n [0.001 Hz] = ( ( v [µm/s] / 1 ) / (pi * ( diam [mm] / 1 ) ) ) * 1
	// 								 = v [µm/s] / (pi * diam [mm])
	IF ( diam_mm = 0.0 ) THEN
		IF ( FIXED_DIAM = 0.0 ) THEN
			// Invalid input for FIXED_DIAM, return velocity setpoint = 0.0
			diam_mm		:= 1.0;
			veloM		:= 0.0;
		ELSE
			// Invalid input for diam_mm, calculate with FIXED_DIAM
			diam_mm		:= FIXED_DIAM;
		END_IF
	END_IF
	UtilCalcSetVeloHz		:= veloM / ( MATH_PI * diam_mm );

END_FUNCTION
```

#### UtilGetVeloHz.st - Calculate velocity in user units [0.001 Hz] from input velocity in user units [µm/s]
```iecst
(********************************************************************
 * COPYRIGHT -- Bernecker + Rainer
 ********************************************************************
 * Library: UtilTyp
 * File: UtilGetVeloHz.st
 * Author: schoenefeldr
 * Created: August 02, 2012
 ********************************************************************
 * Implementation of library UtilTyp
 ********************************************************************)

(* Calculate velocity in user units [0.001 Hz] from input velocity in user units [µm/s] *)
FUNCTION UtilGetVeloHz
	// Formula:
	// 					n [0.001 Hz] = ( v / (pi * diam [mm]) ) * 1.000
	// normalized		n [0.001 Hz] = ( ( v / 1.000.000 ) / (pi * ( diam [mm] / 1.000 ) ) ) * 1.000
	// reduced:			n [0.001 Hz] = ( ( v / 1.000 ) / (pi * ( diam [m] / 1.000 ) ) ) * 1
	// finally reduced:	n [0.001 Hz] = ( ( v / 1 ) / (pi * ( diam [m] / 1 ) ) ) * 1
	// 								 = v / (pi * diam [m])
	// If diameter = 0.0 (invalid diameter) then return 0.0
	IF ( diam_mm = 0.0 ) THEN
		UtilGetVeloHz		:= 0.0;
	ELSE
		UtilGetVeloHz		:= veloM / ( MATH_PI * diam_mm );
	END_IF

END_FUNCTION
```

#### UtilScal.st - Scaling an input via a line equation
```iecst
(********************************************************************
 * COPYRIGHT -- Bernecker + Rainer
 ********************************************************************
 * Library: UtilTyp
 * File: UtilScal.st
 * Author: schoenefeldr
 * Created: September 19, 2012
 ********************************************************************
 * Implementation of library UtilTyp
 ********************************************************************)

(* Scaling an input via a line equation *)
FUNCTION UtilScal
	// This function has a comparable functionality as LCRScal from the CoopConR Lib.
	// As long as the Lib is not necessary this function replaces the Function Block
	UtilScal	:= Gain * In + Offset;
END_FUNCTION
```

### Library Logical/Libraries/UserSpilke (IEC, version 1.06.0) - Spilker specific function blocks
Depends on: AsMath, Acp10_MC

#### UserSpilke.typ - Exported data types
```iecst
(********************************************************************
 * COPYRIGHT -- Bernecker + Rainer
 ********************************************************************
 * Library: UserSpilke
 * File: UserSpilke.typ
 * Author: knausenbergl
 * Created: November 09, 2012
 ********************************************************************
 * Data types of library UserSpilke
 ********************************************************************)

TYPE
	SPR_AUT_PAR_TYP : 	STRUCT
		StartMasterVelocity : REAL; (*Master velocity at very first cut [Master Units/ s]*)
		MaxMasterVelocity : REAL; (*Maximum master velocity [Master Units/ s]*)
		Insetting : REAL; (*Insetting ratio for calculation of CutRangeMaster [%]*)
		MaxCorrection : DINT; (*Maximum correction movement per product cycle [Master Units]*)
		CutStartPos : DINT; (*Start of synchronisation within slave period [Slave Units]*)
		CutEndPos : DINT; (*End of synchronisation within slave period [Slave Units]*)
		MinCutRangeSlave : REAL; (*Minimum synchronization distance [Slave Units]*)
		MinCompRangeSlave : REAL; (*Minimum effective compensation distance [Slave Units]*)
	END_STRUCT;
	SPR_SYNC_PAR_TYP : 	STRUCT
		Velocity : REAL; (*Velocity for reaching phase shift [Master Units / s²]*)
		Acceleration : REAL; (*Acceleration for reaching phase shift [Master Units / s²]*)
	END_STRUCT;
	SPR_PUNCH_IS_TYP : 	STRUCT
		OffsetValue1 : DINT; (*cumulated offset correction*)
		OffsetValue : DINT; (*cumulated offset correction*)
		CutCntOld : UDINT;
		OffsetErrorValid : BOOL;
		PositionErrorValid : BOOL;
		PositionError : DINT;
		R_TRIG_Enable : R_TRIG;
		R_TRIG_Sync : R_TRIG;
		R_TRIG_InCompensation : R_TRIG;
		SPR_RmCapture_0 : SPR_RmCapture; (*RegMark detection*)
		MC_BR_Phasing_0 : MC_BR_Phasing; (*Synchronization movement*)
		MC_BR_CrossCutterControl_0 : MC_BR_CrossCutterControl; (*Cam automat*)
		MC_MoveAbsolute_0 : MC_MoveAbsolute; (*Setup movement before coupling*)
		MC_BR_ReadAutPosition_0 : MC_BR_ReadAutPosition; (*Reading of actual automat position for restart*)
		MC_ReadParameter_AxisPeriod : MC_ReadParameter; (*Reading of axis period for setup movement*)
		LCRLimit_Correction : LCRLimit; (*Limit RM correction movement*)
		RelativeShift : DINT; (*Relative shift for RM correction*)
		State : emuSPR_Punch_State;
		EnableRestart : BOOL; (*Enable cam automat restart*)
		MC_ReadActualPosition_0 : MC_ReadActualPosition;
		ShiftInProgress : BOOL;
		NeutralPosition : REAL; (*Neutral position where axis is not in synchronisation*)
		LCRLimScal_CutRangeMaster : LCRLimScal;
		SPR_RmCalcPosError_Virtual : SPR_RmCalcPosError; (*Calculate position error for virtual registration marks*)
		CutCount_1 : UDINT;
		CccTriggerInit : BOOL; (*Trigger inititalization of CCC*)
		CccInitMasterMaxVel : BOOL; (*Init max. master velocity*)
	END_STRUCT;
	SPR_JOGGEAR_IS_TYP : 	STRUCT
		MC_Halt_0 : MC_Halt;
		MC_GearIn_0 : MC_GearIn;
		MC_ReadStatus_0 : MC_ReadStatus;
		State : USINT;
		R_TRIG_Jog : R_TRIG;
		GearRatioChanged : BOOL;
	END_STRUCT;
	SPR_SETUP_PAR_TYP : 	STRUCT
		Velocity : REAL; (*Maximum velocity [Slave Units / s]*)
		Acceleration : REAL; (*Maximum acceleration [Slave Units / s²]*)
		Deceleration : REAL; (*Maximum deceleration [Slave Units / s²]*)
	END_STRUCT;
	SPR_REG_MARK_PAR_TYP : 	STRUCT
		Axis : UDINT; (*Axis object of Touchprobe*)
		TriggerInput : MC_BR_TRIGGER_REF; (*Input that is used as event source*)
		DistanceToSensor : DINT; (*Distance between tool and sensor [Master Units]*)
		RegMarkPosition : DINT; (*RegMark offset relative to cut position [Master Units]*)
		WindowNegative : REAL; (*Range before the expected position in which the trigger signal may occur [Master Units]*)
		WindowPositive : REAL; (*Range after the expected position in which the trigger signal may occur [Master Units]*)
		EnableRmCorrection : BOOL; (*Enable RM correction*)
		EnableVRegMark : BOOL; (*Use virtual reg mark instead of physical sensor signal*)
		EnableOffsetCorr : BOOL; (*Allow longitudinal correction of register*)
	END_STRUCT;
	basic_status_typ : 	STRUCT  (*status structure*)
		ErrorID : UINT; (*ErrorID of any occured error*)
		ErrorText : ARRAY[0..3]OF STRING[79]; (*Error Text*)
		ActPosition : REAL; (*actual position of the axis*)
		ActVelocity : REAL; (*actual velocity of the axis*)
		DriveStatus : MC_DRIVESTATUS_TYP; (*actual status of the axis*)
	END_STRUCT;
	basic_axisState_typ : 	STRUCT  (*axis state structure*)
		Disabled : BOOL; (*if set, axis is in state Disabled*)
		StandStill : BOOL; (*if set, axis is in state StandsStill*)
		Homing : BOOL; (*if set, axis is in state Homing*)
		Stopping : BOOL; (*if set, axis is in state Stopping*)
		DiscreteMotion : BOOL; (*if set, axis is in state DiscreteMotion*)
		ContinuousMotion : BOOL; (*if set, axis is in state ContinousMotion*)
		SynchronizedMotion : BOOL; (*if set, axis is in state SynchronizedMotion*)
		ErrorStop : BOOL; (*if set, axis is in state ErrorStop*)
		Homed : BOOL;
	END_STRUCT;
	basic_typ : 	STRUCT  (*control structure*)
		Command : basic_command_typ; (*command structure*)
		Parameter : basic_parameter_typ; (*parameter structure*)
		Status : basic_status_typ; (*status structure*)
		AxisState : basic_axisState_typ; (*axis state structure*)
	END_STRUCT;
	emuSPR_Punch_State :
		(
		SPR_STATE_DISABLED,
		SPR_STATE_INIT,
		SPR_STATE_IDLE,
		SPR_STATE_CHECK_STANDBY,
		SPR_STATE_READ_AUT_POS,
		SPR_STATE_MOVE_TO_AUT_POS,
		SPR_STATE_MOVE_TO_NEUTRAL_POS,
		SPR_STATE_W4_REG_MARK,
		SPR_STATE_START_AUTOMAT,
		SPR_STATE_RUNNING,
		SPR_STATE_W4_RESET,
		SPR_STATE_ERROR
		);
	basic_command_typ : 	STRUCT  (*command structure*)
		Power : BOOL; (*switch on the controller*)
		Home : BOOL; (*reference the axis*)
		MoveAbsolute : BOOL; (*move to an defined position*)
		MoveAdditive : BOOL; (*move a defiened distance*)
		MoveVelocity : BOOL; (*start a movement with a defiened velocity*)
		Halt : BOOL; (*stop every active movement*)
		Stop : BOOL; (*stop every active movement as long as is set*)
		MoveJogPos : BOOL; (*move in positive direction as long as is set*)
		MoveJogNeg : BOOL; (*move in negative direction as long as is set*)
		ErrorAcknowledge : BOOL; (*reset active errors*)
	END_STRUCT;
	basic_parameter_typ : 	STRUCT  (*parameter structure*)
		Position : REAL; (*target-position for MoveAbsolute-Command*)
		Distance : REAL; (*distance for MoveAdditive-Command*)
		Velocity : REAL; (*velocity for MoveVelocity-Command*)
		Direction : USINT; (*direction for commanded movements*)
		Acceleration : REAL; (*acceleration for commanded movements*)
		Deceleration : REAL; (*deceleration for commanded movements*)
		HomePosition : REAL; (*target-position for referencing the axis*)
		HomeMode : USINT; (*homing mode*)
		JogVelocity : REAL; (*velocity for jogging movement*)
	END_STRUCT;
END_TYPE
```

#### UserSpilke.fun - Exported functions and function blocks
```iecst
(********************************************************************
 * COPYRIGHT -- Bernecker + Rainer
 ********************************************************************
 * Library: UserSpilke
 * File: UserSpilke.fun
 * Author: knausenbergl
 * Created: November 09, 2012
 ********************************************************************
 * Functions and function blocks of library UserSpilke
 ********************************************************************)

FUNCTION_BLOCK SPR_PneumLever (*pneumatic lever (unwinder up down)*)
	VAR_INPUT
		Up : BOOL; (*move up command*)
		Down : BOOL; (*move down command*)
		LimitSwitchTop : BOOL; (*limitswich top*)
		LimitSwitchBottom : BOOL; (*limitswitch bottom*)
	END_VAR
	VAR_OUTPUT
		ValveUp : BOOL; (*switch on valve (to move upwards)*)
		ValveDown : BOOL; (*switch on valve (to move downwards)*)
	END_VAR
END_FUNCTION_BLOCK

FUNCTION_BLOCK SPR_Punch (*Implements the punch operation in automatic mode*)
	VAR_INPUT
		Master : UDINT; (*Master axis reference*)
		Slave : UDINT; (*Slave axis reference*)
		Enable : BOOL;
		EnableMove : BOOL; (*Allow this FUB to execute movements*)
		SearchRM : BOOL; (*Initiate search of new RM on positive edge*)
		RestartAllowed : BOOL; (*Execute a synchronization movement (only possible when "Move" is TRUE)*)
		Sync : BOOL; (*Execute a synchronization movement (only possible when "Move" is TRUE)*)
		VRmCorrection : DINT; (*Correction value for virtual marks*)
		ProductLength : DINT; (*Product length [Master Units]*)
		VRmRecordedPosition : DINT; (*Recorded position when using virtual registration mark*)
		RegMarkPar : SPR_REG_MARK_PAR_TYP; (*Parameters for registration mark detection and evaluation*)
		AutPar : SPR_AUT_PAR_TYP; (*Cam automat parameters*)
		SyncPar : SPR_SYNC_PAR_TYP; (*Parameters for the synchronization movement*)
		SetupPar : SPR_SETUP_PAR_TYP; (*Parameters for setting up the axis before coupling*)
	END_VAR
	VAR_OUTPUT
		Active : BOOL; (*Cam automat is running*)
		Error : BOOL;
		ErrorID : UINT;
		EnableRestart : BOOL;
		SetupComplete : BOOL; (*Setup movement complete, punch clamp can be closed*)
		CutMasterPosition : DINT; (*Cut master position [Master Units]*)
		ProbeCounter : UDINT; (*Counter for valid trigger events*)
		MissedTriggers : UDINT; (*Counter for missed trigger events*)
		ActPositionError : DINT; (*Actual reg mark position error [Master Units]*)
	END_VAR
	VAR
		IS : SPR_PUNCH_IS_TYP;
	END_VAR
END_FUNCTION_BLOCK

FUNCTION_BLOCK SPR_HydLever (*Hydraulic lever (e.g. of the unwinder)*)
	VAR_INPUT
		Up : BOOL; (*move up command*)
		Down : BOOL; (*move down command*)
		LimitSwitchTop : BOOL;
		LimitSwitchBottom : BOOL;
	END_VAR
	VAR_OUTPUT
		ValveOn : BOOL; (*switch on valve (to move downwards)*)
		MotorOn : BOOL; (*switch on motor*)
	END_VAR
END_FUNCTION_BLOCK

FUNCTION_BLOCK SPR_WinderClutch (*Control of prop. valve for winder clutch*)
	VAR_INPUT
		RefDiameter : ARRAY[0..1] OF REAL; (*reference diameters [Master Units]
RefDiameter[0] = diameter at min. pressure
RefDiameter[1] = diameter at max. pressure*)
		RefPressure : ARRAY[0..1] OF REAL; (*reference pressure [%]
RefPressure[0] = min. pressure
RefPressure[1] = max. pressure*)
		ActDiameter : REAL; (*actual winder diameter [Master Units]*)
	END_VAR
	VAR_OUTPUT
		SetPressure : REAL; (*set valve pressure [%]*)
	END_VAR
	VAR
		LCRLimScal_Pressure : LCRLimScal;
	END_VAR
END_FUNCTION_BLOCK

FUNCTION_BLOCK SPR_CheckTextIndexValid (*Checks if a textgroup index exists*)
	VAR_INPUT
		Enable : BOOL;
		VCHandle : UDINT;
		TG_id : UDINT;
		TGT_id : UINT;
	END_VAR
	VAR_OUTPUT
		Status : UINT;
		Valid : BOOL;
		Text : STRING[80];
	END_VAR
	VAR
		TextLength : UINT;
	END_VAR
END_FUNCTION_BLOCK

FUNCTION_BLOCK SPR_MeterCounter (*Counts length periods on an axis*)
	VAR_INPUT
		Enable : BOOL; (*Enables the cam switch*)
		Period : REAL; (*Definition of the period, in case a non-periodic master axis is used or if the cam switch period does not match the master axis period*)
		Axis : UDINT; (*Axis reference of the axis from which the position is being taken*)
	END_VAR
	VAR_OUTPUT
		InOperation : BOOL; (*The controlled track is enabled.*)
		Busy : BOOL; (*FB is not yet finished*)
		Error : BOOL; (*Error occurred in FB*)
		ErrorID : UINT; (*Error number*)
	END_VAR
	VAR_IN_OUT
		PeriodCount : UDINT; (*Period count (incremented every time the axis moves another period)*)
	END_VAR
	VAR
		MC_BR_DigitalCamSwitch_0 : MC_BR_DigitalCamSwitch;
		F_TRIG_Value : F_TRIG;
	END_VAR
END_FUNCTION_BLOCK

FUNCTION_BLOCK SPR_ScaleCircumference (*Scales a tool circumference to a whole number that is divisible without remainder by the number of tool segments*)
	VAR_INPUT
		ActCircumference : REAL;
		NumberToolSegments : USINT;
	END_VAR
	VAR_OUTPUT
		ScaledCircumference : UDINT;
		ToolSegmentPeriod : UDINT;
	END_VAR
	VAR
		Remainder : DINT;
	END_VAR
END_FUNCTION_BLOCK

FUNCTION_BLOCK SPR_DrivesGlobal (*Monitors the status of all drives*)
	VAR_INPUT
		Init : BOOL; (*Allocates memory for the required number of function blocks*)
		Enable : BOOL; (*Enables function block*)
		pAxes : UDINT; (*Pointer to UDINT array with axis objects*)
		MaxNumberAxes : USINT; (*Maximum number of axis objects*)
	END_VAR
	VAR_OUTPUT
		InitDone : BOOL; (*Memory successfully allocated*)
		Valid : BOOL;
		Busy : BOOL;
		Error : BOOL;
		ErrorID : UINT;
		DriveStatusAll : MC_DRIVESTATUS_TYP; (*DriveStatus[Axis_1] AND DriveStatus[Axis_2] AND ... AND DriveStatus[Axis_N]*)
		DriveStatusAny : MC_DRIVESTATUS_TYP; (*DriveStatus[Axis_1] OR DriveStatus[Axis_2] OR ... OR DriveStatus[Axis_N]*)
	END_VAR
	VAR
		pMC_BR_ReadDriveStatus : REFERENCE TO MC_BR_ReadDriveStatus;
		State : USINT;
		StartAddress : UDINT; (*start address of dynamic MC_BR_ReadDriveStatus array*)
		pAxis : REFERENCE TO UDINT;
		C_MaxNumberAxes : USINT;
		MC_BR_ReadDriveStatus_Dummy : ARRAY[0..0] OF MC_BR_ReadDriveStatus;
		AllocStatus : UINT; (*status of TMP_Alloc function*)
		AxisIndex : USINT;
		TempDriveStatus : MC_DRIVESTATUS_TYP;
	END_VAR
END_FUNCTION_BLOCK

FUNCTION_BLOCK SPR_MoveMaster (*Starts a movement of the master axis*)
	VAR_INPUT
		Enable : BOOL;
		SlavesReady : BOOL;
		AdditiveMovement : BOOL;
		Velocity : BOOL;
		Acceleration : BOOL;
		Deceleration : BOOL;
		Distance : BOOL;
	END_VAR
	VAR_OUTPUT
		Error : BOOL;
		ErrorID : UINT;
		Busy : BOOL;
	END_VAR
	VAR
		MC_Halt : MC_Halt;
		New_Member : MC_BR_JogVelocity;
	END_VAR
END_FUNCTION_BLOCK

FUNCTION_BLOCK SPR_UnwinderCtrl (*Controls an unwinder with a magnet particle brake*)
	VAR_INPUT
		Enable : BOOL;
		InitPidPar : BOOL; (*Initialize PID parameters on positive edge*)
		PidPar : wnc_pidPara_typ; (*PID controller parameters*)
		CoreInertia : REAL; (*Mass moment of inertia of empty winder [kgm²]*)
		CoreDiam : REAL; (*Diameter of empty winder [m]*)
		MaxDiam : REAL; (*Maximum winder diameter [m]*)
		MaxRollMass : REAL; (*Mass of roll at maximum diameter [kg]*)
		ForceFf : REAL; (*Feed forward force [N]*)
		ActDiam : REAL; (*Actual winder diameter [m]*)
		SetDancerPos : REAL; (*Set dancer position [Dancer Units]*)
		ActDancerPos : REAL; (*Actual dancer position [Dancer Units]*)
		MaxTorque : REAL; (*Maximum brake torque [Nm]*)
	END_VAR
	VAR_OUTPUT
		Status : UINT;
		SetTorque : REAL; (*Set torque for winder brake*)
	END_VAR
	VAR
		State : USINT;
		WNCPidCtrl_0 : WNCPidCtrl;
		K_RollMass : REAL; (*Constant to calculate actual mass of Roll: K_RollMass = Pi * MaterialWidth * MaterialDensity*)
		ActRollMass : REAL;
		ActInertia : REAL;
	END_VAR
END_FUNCTION_BLOCK

FUNCTION_BLOCK SPR_LabelerAut (*Cam automat configuration for labeling unit*)
	VAR_INPUT
		Master : UDINT; (*Master axis object*)
		LabelPeriod : REAL; (*Label period [Units]*)
		DistanceToLabelSensor : REAL; (*Distance between sensor and labelling position [Units]*)
		MaxMasterVelocity : REAL; (*Maximum master velocity [Units / s]*)
		ProductLengthMaster : REAL; (*Product length on master axis [Units]*)
		TriggerEvent : USINT; (*Trigger event for correction, e.g. ncTrigger1 + ncP_EDGE*)
	END_VAR
	VAR_OUTPUT
		adrAutData : UDINT;
	END_VAR
	VAR
		AutData : MC_AUTDATA_TYP;
	END_VAR
END_FUNCTION_BLOCK

FUNCTION_BLOCK SPR_LabelerAutVax (*Cam automat configuration for an "ideal" labeler (no label position correction)*)
	VAR_INPUT
		Master : UDINT; (*Master axis object*)
		LabelPeriod : REAL; (*Label period [Units]*)
		ProductLengthMaster : REAL; (*Product length on master axis [Units]*)
		DistanceToRmSensor : REAL; (*Distance between sensor and labelling position [Units]*)
		MaxMasterVelocity : REAL; (*Maximum master velocity [Units / s]*)
		RegMarkPosition : REAL; (*Reg mark position relative to label [Units]*)
		CamLength : REAL; (*Distance the label runs synchronized to master [Units]*)
		CorrectionLongitudinal : BOOL; (*Manually longitudinal correction*)
		CorrectionLongitudinalValue : REAL; (*Manually longitudinal correction value*)
		AccelerationBias : REAL; (*AccelerationDistance / DecelerationDistance
Valid Range: 0.1...10.0
<0.1   ...   AccelerationDistance = DecelerationDistance (default)
0.1     ...   AccelerationDistance = 0.1 * DecelerationDistance
1.0     ...   AccelerationDistance = DecelerationDistance
2.0     ...   AccelerationDistane   = DecelerationDistance
10.0   ...   AccelerationDistance = 10 * DecelerationDistance
>10.0 ...   AccelerationDistance = DecelerationDistance (default)*)
		TriggerEvent : USINT; (*Trigger event for correction, e.g. ncTrigger1 + ncP_EDGE*)
	END_VAR
	VAR_OUTPUT
		adrAutData : UDINT;
	END_VAR
	VAR
		AutData : MC_AUTDATA_TYP;
		AccelerationDistance : REAL;
		DecelerationDistance : REAL;
	END_VAR
END_FUNCTION_BLOCK

FUNCTION_BLOCK SPR_OverflowDetection (*Detects overflow e,g, of a periodic position*)
	VAR_INPUT
		PeriodicPosition : DINT; (*Periodic position*)
		ModuloPeriod : DINT; (*Modulo period at which overflow occurs*)
		Enable : BOOL; (*Enables FUB*)
	END_VAR
	VAR_OUTPUT
		AbsolutePosition : DINT; (*Absolute position (reset when FUB is disabled)*)
		PositiveOverflow : BOOL; (*Overflow in negative direction (TRUE for 1 cycle)*)
		NegativeOverflow : BOOL; (*Overflow in positive direction (TRUE for 1 cycle)*)
	END_VAR
	VAR
		PeriodOffset : DINT; (*Offset of actual period*)
		PeriodicPosition_1 : DINT;
		R_TRIG_Enable : R_TRIG;
	END_VAR
END_FUNCTION_BLOCK

FUNCTION_BLOCK SPR_JogGear (*Gear in and update the gear ratio as long as the Jog input is set*)
	VAR_INPUT
		Jog : BOOL;
		Master : UDINT;
		Slave : UDINT;
		RatioNumerator : INT;
		RatioDenominator : UINT;
		Acceleration : REAL;
		Deceleration : REAL;
		MasterParID : UINT;
		MasterParIDMaxVelocity : REAL;
	END_VAR
	VAR_OUTPUT
		InGear : BOOL;
		Halting : BOOL;
		Busy : BOOL;
		CommandAborted : BOOL;
		Error : BOOL;
		ErrorID : UINT;
	END_VAR
	VAR
		IS : SPR_JOGGEAR_IS_TYP;
	END_VAR
END_FUNCTION_BLOCK

FUNCTION_BLOCK FB_LaminateCTRL (*TODO: Bitte Kommentar hier einzufügen*)
	VAR_IN_OUT
		machineMaster : USINT; (*SPR_MoveMaster;(*ACP10AXIS_typ;*)
		status : USINT; (*unitAxis 		:FB_AxisCtrl;*)
		MarkpointMaster : SPR_RmCapture;
		MarkpointUnit : SPR_RmCapture;
		State : emuSPR_Punch_State;
		newParam5 : BOOL;
	END_VAR
	VAR
		StateCtrl : INT;
	END_VAR
	VAR CONSTANT
		STATE_READY : USINT := 10;
		STATE_POWER_ON : USINT := 1;
		STATE_MOVE_VELOCITY : USINT := 16;
		STATE_MOVE_ABSOLUTE : USINT := 14;
		STATE_WAIT : USINT := 0;
		STATE_STOP : USINT := 11;
		STATE_MOVE_ADDITIVE : USINT := 15;
		STATE_HOME : USINT := 2;
		STATE_ERROR_RESET : USINT := 102;
		STATE_ERROR_AXIS : USINT := 100;
		STATE_ERROR : USINT := 101;
		STATE_JOG_POSITIVE : USINT := 12;
		STATE_JOG_NEGATIVE : USINT := 13;
		STATE_HALT : USINT := 17;
	END_VAR
END_FUNCTION_BLOCK
(*
FUNCTION_BLOCK FB_AxisCtrl
	VAR_INPUT
		BasicControl 			:basic_typ;
		MC_Home_0 				:MC_Home;
		MC_MoveAbsolute_0 		:MC_MoveAbsolute;
		MC_MoveAdditive_0 		:MC_MoveAdditive;
		MC_MoveVelocity_0 		:MC_MoveVelocity;
		MC_Power_0 				:MC_Power;
		MC_ReadActualPosition_0 : MC_ReadActualPosition;
		MC_ReadActualVelocity_0 : MC_ReadActualVelocity;
		MC_ReadAxisError_0 		: MC_ReadAxisError;
		MC_ReadStatus_0 		: MC_ReadStatus;
		MC_Reset_0 				: MC_Reset;
		MC_Stop_0 				: MC_Stop;
		MC_BR_ReadDriveStatus_0 : MC_BR_ReadDriveStatus;
		MC_Halt_0 				: MC_Halt;
		MC_GearIn_0				: MC_GearIn;
		Axis1Obj 				: UDINT;
		AxisStep 				: UINT;
	END_VAR
	VAR CONSTANT
		STATE_READY 		: USINT := 10;
		STATE_POWER_ON		: USINT := 1;
		STATE_MOVE_VELOCITY : USINT := 16;
		STATE_MOVE_ABSOLUTE : USINT := 14;
		STATE_WAIT 			: USINT := 0;
		STATE_STOP 			: USINT := 11;
		STATE_MOVE_ADDITIVE : USINT := 15;
		STATE_HOME 			: USINT := 2;
		STATE_ERROR_RESET 	: USINT := 102;
		STATE_ERROR_AXIS 	: USINT := 100;
		STATE_ERROR 		: USINT := 101;
		STATE_JOG_POSITIVE 	: USINT := 12;
		STATE_JOG_NEGATIVE 	: USINT := 13;
		STATE_HALT 			: USINT := 17;
	END_VAR
END_FUNCTION_BLOCK
*)

FUNCTION_BLOCK FB_MainCtrl (*TODO: Bitte Kommentar hier einzufügen*)
	VAR_INPUT
		cycletime : UDINT;
		mainCtrlState : USINT;
		rcpActState : USINT;
	END_VAR
END_FUNCTION_BLOCK
(*FUNCTION_BLOCK FB_MainHw  (*TODO: Bitte Kommentar hier einzufügen*)
(*	VAR_INPUT
		SL8010_8A1 :   BOOL ;  (**)
(*		SO4110_38A5 :   BOOL ;  (**)
(*	END_VAR
END_FUNCTION_BLOCK*)

FUNCTION_BLOCK FB_MainHW (*TODO: Bitte Kommentar hier einzufügen*)
	VAR_INPUT
		SL8010_8A1 : BOOL;
		SO4110_38A5 : BOOL;
	END_VAR
END_FUNCTION_BLOCK
```

#### SPR_HydLever.st - Hydraulic lever (e.g. of the unwinder)
```iecst
(********************************************************************
 * COPYRIGHT -- Bernecker + Rainer
 ********************************************************************
 * Library: UserSpilke
 * File: SPR_HydLever.st
 * Author: knausenbergl
 * Created: November 15, 2012
 ********************************************************************
 * Implementation of library UserSpilke
 ********************************************************************)

(*<$Description$> Hydraulic lever (e.g. of the unwinder) </$Description$>*)
FUNCTION_BLOCK SPR_HydLever
	ValveOn	:= Down AND NOT Up;
	MotorOn	:= NOT LimitSwitchTop AND Up AND NOT Down;
END_FUNCTION_BLOCK
```

#### SPR_WinderClutch.st - Control of prop. valve for winder clutch
```iecst
(********************************************************************
 * COPYRIGHT -- Bernecker + Rainer
 ********************************************************************
 * Library: UserSpilke
 * File: SPR_Spender.st
 * Author: knausenbergl
 * Created: November 20, 2012
 ********************************************************************
 * Implementation of library UserSpilke
 ********************************************************************)

(*<$Description$> Control of prop. valve for winder clutch </$Description$>*)
FUNCTION_BLOCK SPR_WinderClutch
	LCRLimScal_Pressure.x1	:= RefDiameter[0];
	LCRLimScal_Pressure.x2	:= RefDiameter[1];
	LCRLimScal_Pressure.y1	:= LIMIT(0.0, RefPressure[0], 100.0);
	LCRLimScal_Pressure.y2	:= LIMIT(0.0, RefPressure[1], 100.0);
	LCRLimScal_Pressure.x	:= ActDiameter;
	LCRLimScal_Pressure();
	SetPressure	:= LCRLimScal_Pressure.y;
END_FUNCTION_BLOCK
```

#### SPR_CheckTextIndexValid.st - Checks if a textgroup index exists
```iecst
(********************************************************************
 * COPYRIGHT -- Bernecker + Rainer
 ********************************************************************
 * Library: UserSpilke
 * File: SPR_CheckTextIndexValid.st
 * Author: knausenbergl
 * Created: November 23, 2012
 ********************************************************************
 * Implementation of library UserSpilke
 ********************************************************************)

(*<$Description$> Checks if a textgroup index exists </$Description$>*)
FUNCTION_BLOCK SPR_CheckTextIndexValid

	Status	:= VA_Saccess(Enable, VCHandle);
	IF (Status = ERR_OK) THEN
		TextLength	:= SIZEOF(Text);
		Status		:= VA_GetTextByTextGroup(TRUE, VCHandle, TG_id, TGT_id, ADR(Text), ADR(TextLength) );
		Valid		:= (Status = ERR_OK);
		VA_Srelease(TRUE, VCHandle);
	ELSE
		Valid	:= FALSE;
	END_IF;

END_FUNCTION_BLOCK
```

#### SPR_MeterCounter.st - Counts length periods on an axis
```iecst
(********************************************************************
 * COPYRIGHT -- Bernecker + Rainer
 ********************************************************************
 * Library: UserSpilke
 * File: SPR_MeterCounter.st
 * Author: knausenbergl
 * Created: December 06, 2012
 ********************************************************************
 * Implementation of library UserSpilke
 ********************************************************************)

(*<$Description$> Counts length periods on an axis </$Description$>*)
FUNCTION_BLOCK SPR_MeterCounter
	MC_BR_DigitalCamSwitch_0.Switches.Master	:= Axis;
	MC_BR_DigitalCamSwitch_0.OutputOptions.Axis	:= Axis;
	MC_BR_DigitalCamSwitch_0.Switches.Period	:= Period;
	MC_BR_DigitalCamSwitch_0.Switches.Switches[0].FirstOnPosition[0]	:= Period / 2.0;
	MC_BR_DigitalCamSwitch_0.Switches.Switches[0].LastOnPosition[0]		:= Period;
	MC_BR_DigitalCamSwitch_0.EnableValue	:= TRUE;
	MC_BR_DigitalCamSwitch_0.Enable			:= Enable;
	MC_BR_DigitalCamSwitch_0();

	F_TRIG_Value.CLK	:= MC_BR_DigitalCamSwitch_0.Value;
	F_TRIG_Value();

	Error		:= MC_BR_DigitalCamSwitch_0.Error;
	ErrorID		:= MC_BR_DigitalCamSwitch_0.ErrorID;
	Busy		:= MC_BR_DigitalCamSwitch_0.Busy;
	InOperation	:= MC_BR_DigitalCamSwitch_0.InOperation;
	IF (F_TRIG_Value.Q AND MC_BR_DigitalCamSwitch_0.Busy) THEN
		PeriodCount	:= PeriodCount + 1;
	END_IF;
END_FUNCTION_BLOCK
```

#### SPR_ScaleCircumference.st - Scales a tool circumference to a whole number that is divisible without remainder by the number of tool segments
```iecst
(********************************************************************
 * COPYRIGHT -- Bernecker + Rainer
 ********************************************************************
 * Library: UserSpilke
 * File: SPR_ScaleCircumference.st
 * Author: knausenbergl
 * Created: December 07, 2012
 ********************************************************************
 * Implementation of library UserSpilke
 ********************************************************************)

(*<$Description$> Scales a tool circumference to a whole number that is divisible without remainder by the number of tool segments </$Description$>*)
FUNCTION_BLOCK SPR_ScaleCircumference
	IF (NumberToolSegments > 0) THEN
		Remainder	:= REAL_TO_DINT(floor(ActCircumference) ) MOD USINT_TO_DINT(NumberToolSegments);

		IF (Remainder > USINT_TO_DINT(NumberToolSegments / 2) ) THEN
			Remainder	:= Remainder - USINT_TO_DINT(NumberToolSegments);
		END_IF;

		ScaledCircumference	:= DINT_TO_UDINT(REAL_TO_DINT(floor(ActCircumference) ) - Remainder);
		ToolSegmentPeriod	:= ScaledCircumference / NumberToolSegments;
	ELSE
		ScaledCircumference	:= 0;
		ToolSegmentPeriod	:= 0;
	END_IF;

END_FUNCTION_BLOCK
```

#### SPR_DrivesGlobal.st - Monitors the status of all drives
```iecst
(********************************************************************
 * COPYRIGHT -- Bernecker + Rainer
 ********************************************************************
 * Library: UserSpilke
 * File: DrivesGlobal.st
 * Author: knausenbergl
 * Created: December 13, 2012
 ********************************************************************
 * Implementation of library UserSpilke
 ********************************************************************)

(*<$Description$> Monitors the status of all drives </$Description$>*)
FUNCTION_BLOCK SPR_DrivesGlobal
	CASE State OF
		//IDLE, waiting for init command
		0:
			IF (Init AND (MaxNumberAxes <> 0) AND (pAxes <> 0) ) THEN
				AllocStatus	:= TMP_alloc( (SIZEOF(MC_BR_ReadDriveStatus_Dummy[0]) * MaxNumberAxes), ADR(StartAddress) );
				InitDone	:= (AllocStatus = 0);
				IF (InitDone) THEN
					memset(StartAddress, 0, (SIZEOF(MC_BR_ReadDriveStatus_Dummy[0]) * MaxNumberAxes) );
					C_MaxNumberAxes	:= MaxNumberAxes;
					State			:= 1;
				END_IF;
			END_IF;

		//INIT COMPLETE, waiting for enable command
		1:
			IF (Enable AND (pAxes <> 0) ) THEN
				Valid	:= TRUE;
				Busy	:= FALSE;
				Error	:= FALSE;
				ErrorID	:= 0;

				DriveStatusAll.AxisError		:= TRUE;
				DriveStatusAll.ControllerReady	:= TRUE;
				DriveStatusAll.ControllerStatus	:= TRUE;
				DriveStatusAll.DriveEnable		:= TRUE;
				DriveStatusAll.HomeSwitch		:= TRUE;
				DriveStatusAll.HomingOk			:= TRUE;
				DriveStatusAll.LagWarning		:= TRUE;
				DriveStatusAll.NegHWSwitch		:= TRUE;
				DriveStatusAll.NetworkInit		:= TRUE;
				DriveStatusAll.PosHWSwitch		:= TRUE;
				DriveStatusAll.ResetDone		:= TRUE;
				DriveStatusAll.Simulation		:= TRUE;
				DriveStatusAll.Trigger1			:= TRUE;
				DriveStatusAll.Trigger2			:= TRUE;

				DriveStatusAny.AxisError		:= FALSE;
				DriveStatusAny.ControllerReady	:= FALSE;
				DriveStatusAny.ControllerStatus	:= FALSE;
				DriveStatusAny.DriveEnable		:= FALSE;
				DriveStatusAny.HomeSwitch		:= FALSE;
				DriveStatusAny.HomingOk			:= FALSE;
				DriveStatusAny.LagWarning		:= FALSE;
				DriveStatusAny.NegHWSwitch		:= FALSE;
				DriveStatusAny.NetworkInit		:= FALSE;
				DriveStatusAny.PosHWSwitch		:= FALSE;
				DriveStatusAny.ResetDone		:= FALSE;
				DriveStatusAny.Simulation		:= FALSE;
				DriveStatusAny.Trigger1			:= FALSE;
				DriveStatusAny.Trigger2			:= FALSE;

				FOR AxisIndex	:= 0 TO (C_MaxNumberAxes - 1) DO
					pAxis	ACCESS (pAxes + AxisIndex * SIZEOF(UDINT) );
					pMC_BR_ReadDriveStatus	ACCESS (StartAddress + AxisIndex * SIZEOF(MC_BR_ReadDriveStatus_Dummy[0]) );

					pMC_BR_ReadDriveStatus.AdrDriveStatus	:= ADR(TempDriveStatus);
					pMC_BR_ReadDriveStatus.Axis				:= pAxis;
					pMC_BR_ReadDriveStatus.Enable			:= (pAxis <> 0);
					pMC_BR_ReadDriveStatus();

					IF (pMC_BR_ReadDriveStatus.Enable) THEN
						Valid	:= Valid AND pMC_BR_ReadDriveStatus.Valid;
						Busy	:= Busy OR pMC_BR_ReadDriveStatus.Busy;
						Error	:= Error OR pMC_BR_ReadDriveStatus.Error;
						IF (pMC_BR_ReadDriveStatus.ErrorID <> ERR_OK) THEN
							ErrorID	:= pMC_BR_ReadDriveStatus.ErrorID;
						END_IF;

						DriveStatusAll.AxisError		:= DriveStatusAll.AxisError AND TempDriveStatus.AxisError;
						DriveStatusAll.ControllerReady	:= DriveStatusAll.ControllerReady AND TempDriveStatus.ControllerReady;
						DriveStatusAll.ControllerStatus	:= DriveStatusAll.ControllerStatus AND TempDriveStatus.ControllerStatus;
						DriveStatusAll.DriveEnable		:= DriveStatusAll.DriveEnable AND TempDriveStatus.DriveEnable;
						DriveStatusAll.HomeSwitch		:= DriveStatusAll.HomeSwitch AND TempDriveStatus.HomeSwitch;
						DriveStatusAll.HomingOk			:= DriveStatusAll.HomingOk AND TempDriveStatus.HomingOk;
						DriveStatusAll.LagWarning		:= DriveStatusAll.LagWarning AND TempDriveStatus.LagWarning;
						DriveStatusAll.NegHWSwitch		:= DriveStatusAll.NegHWSwitch AND TempDriveStatus.NegHWSwitch;
						DriveStatusAll.NetworkInit		:= DriveStatusAll.NetworkInit AND TempDriveStatus.NetworkInit;
						DriveStatusAll.PosHWSwitch		:= DriveStatusAll.PosHWSwitch AND TempDriveStatus.PosHWSwitch;
						DriveStatusAll.ResetDone		:= DriveStatusAll.ResetDone AND TempDriveStatus.ResetDone;
						DriveStatusAll.Simulation		:= DriveStatusAll.Simulation AND TempDriveStatus.Simulation;
						DriveStatusAll.Trigger1			:= DriveStatusAll.Trigger1 AND TempDriveStatus.Trigger1;
						DriveStatusAll.Trigger2			:= DriveStatusAll.Trigger2 AND TempDriveStatus.Trigger2;

						DriveStatusAny.AxisError		:= DriveStatusAny.AxisError OR TempDriveStatus.AxisError;
						DriveStatusAny.ControllerReady	:= DriveStatusAny.ControllerReady OR TempDriveStatus.ControllerReady;
						DriveStatusAny.ControllerStatus	:= DriveStatusAny.ControllerStatus OR TempDriveStatus.ControllerStatus;
						DriveStatusAny.DriveEnable		:= DriveStatusAny.DriveEnable OR TempDriveStatus.DriveEnable;
						DriveStatusAny.HomeSwitch		:= DriveStatusAny.HomeSwitch OR TempDriveStatus.HomeSwitch;
						DriveStatusAny.HomingOk			:= DriveStatusAny.HomingOk OR TempDriveStatus.HomingOk;
						DriveStatusAny.LagWarning		:= DriveStatusAny.LagWarning OR TempDriveStatus.LagWarning;
						DriveStatusAny.NegHWSwitch		:= DriveStatusAny.NegHWSwitch OR TempDriveStatus.NegHWSwitch;
						DriveStatusAny.NetworkInit		:= DriveStatusAny.NetworkInit OR TempDriveStatus.NetworkInit;
						DriveStatusAny.PosHWSwitch		:= DriveStatusAny.PosHWSwitch OR TempDriveStatus.PosHWSwitch;
						DriveStatusAny.ResetDone		:= DriveStatusAny.ResetDone OR TempDriveStatus.ResetDone;
						DriveStatusAny.Simulation		:= DriveStatusAny.Simulation OR TempDriveStatus.Simulation;
						DriveStatusAny.Trigger1			:= DriveStatusAny.Trigger1 OR TempDriveStatus.Trigger1;
						DriveStatusAny.Trigger2			:= DriveStatusAny.Trigger2 OR TempDriveStatus.Trigger2;
					END_IF;
				END_FOR;
			ELSE
				Valid	:= FALSE;
				Busy	:= FALSE;
				Error	:= FALSE;
				ErrorID	:= ERR_FUB_ENABLE_FALSE;

				memset(ADR(DriveStatusAll), 0, SIZEOF(DriveStatusAll) );
				memset(ADR(DriveStatusAny), 0, SIZEOF(DriveStatusAny) );

				FOR AxisIndex	:= 0 TO (C_MaxNumberAxes - 1) DO
					pMC_BR_ReadDriveStatus	ACCESS (StartAddress + AxisIndex * SIZEOF(MC_BR_ReadDriveStatus_Dummy[0]) );

					pMC_BR_ReadDriveStatus.AdrDriveStatus	:= ADR(TempDriveStatus);
					pMC_BR_ReadDriveStatus.Axis				:= 0;
					pMC_BR_ReadDriveStatus.Enable			:= FALSE;
					pMC_BR_ReadDriveStatus();
				END_FOR;
			END_IF;

	END_CASE;

END_FUNCTION_BLOCK
```

#### SPR_OverflowDetection.st - Detects overflow e,g, of a periodic position
```iecst
(********************************************************************
 * COPYRIGHT -- Bernecker + Rainer
 ********************************************************************
 * Library: UserSpilke
 * File: OverflowDetection.st
 * Author: knausenbergl
 * Created: February 07, 2013
 ********************************************************************
 * Implementation of library UserSpilke
 ********************************************************************)

(*<$Description$> Detects overflow e,g, of a periodic position </$Description$>*)
FUNCTION_BLOCK SPR_OverflowDetection
	R_TRIG_Enable.CLK	:= Enable;
	R_TRIG_Enable();

	IF (Enable) THEN
		IF (R_TRIG_Enable.Q) THEN
			PeriodicPosition_1	:= PeriodicPosition;	//initialize previous position
		END_IF;

		//detect overflow
		IF (ABS(PeriodicPosition - PeriodicPosition_1) > (ModuloPeriod / 2) ) THEN
			IF (PeriodicPosition < PeriodicPosition_1) THEN
				PositiveOverflow	:= TRUE;
				PeriodOffset		:= PeriodOffset + ModuloPeriod;	//increase period offset
			ELSE
				NegativeOverflow	:= TRUE;
				PeriodOffset		:= PeriodOffset - ModuloPeriod;	//decrease period offset
			END_IF;
		ELSE
			PositiveOverflow	:= FALSE;
			NegativeOverflow	:= FALSE;
		END_IF;

		//absolute position is the sum of offset (from previous periods) and actual periodic position
		AbsolutePosition	:= PeriodOffset + PeriodicPosition;

		//save previous position
		PeriodicPosition_1	:= PeriodicPosition;

	ELSE
		PeriodicPosition_1	:= 0;
		PeriodOffset		:= 0;
		AbsolutePosition	:= 0;
		PositiveOverflow	:= FALSE;
		NegativeOverflow	:= FALSE;
	END_IF;

END_FUNCTION_BLOCK
```

#### SPR_MoveMaster.st - Starts a movement of the master axis
```iecst
(********************************************************************
 * COPYRIGHT -- Bernecker + Rainer
 ********************************************************************
 * Library: UserSpilke
 * File: SPR_MoveMaster.st
 * Author: knausenbergl
 * Created: December 14, 2012
 ********************************************************************
 * Implementation of library UserSpilke
 ********************************************************************)

(*<$Description$> Starts a movement of the master axis </$Description$>*)
FUNCTION_BLOCK SPR_MoveMaster
END_FUNCTION_BLOCK
```

#### SPR_UnwinderCtrl.st - Controls an unwinder with a magnet particle brake
```iecst
(********************************************************************
 * COPYRIGHT -- Bernecker + Rainer
 ********************************************************************
 * Library: UserSpilke
 * File: SPR_UnwinderCtrl.st
 * Author: knausenbergl
 * Created: December 15, 2012
 ********************************************************************
 * Implementation of library UserSpilke
 ********************************************************************)

(*<$Description$> Controls an unwinder with a magnet particle brake </$Description$>*)
FUNCTION_BLOCK SPR_UnwinderCtrl

	CASE State OF

		//********************	DISABLED	********************
		0:
			IF (Enable) THEN
				State	:= 1;
			END_IF;

		//********************	ACTIVE	********************
		1:
			IF (NOT Enable) THEN
				State	:= 0;
			ELSIF ( (WNCPidCtrl_0.status >= 34350) AND (WNCPidCtrl_0.status <= 34449) ) THEN
				State	:= 2;
			END_IF;

		//********************	ERROR	********************
		2:
			IF (NOT Enable) THEN
				State	:= 0;
			END_IF;

	END_CASE;

END_FUNCTION_BLOCK
```

#### SPR_PneumLever.st - Hydraulic lever (e.g. of the unwinder)
```iecst
(********************************************************************
 * COPYRIGHT -- Bernecker + Rainer
 ********************************************************************
 * Library: UserSpilke
 * File: SPR_HydLever.st
 * Author: knausenbergl
 * Created: November 15, 2012
 ********************************************************************
 * Implementation of library UserSpilke
 ********************************************************************)

(*<$Description$> Hydraulic lever (e.g. of the unwinder) </$Description$>*)
FUNCTION_BLOCK SPR_PneumLever
	ValveDown	:= Down AND NOT Up AND NOT LimitSwitchBottom;
	ValveUp		:= Up AND NOT Down AND NOT LimitSwitchTop;
END_FUNCTION_BLOCK
```

#### SPR_JogGear.st - Gear in and update the gear ratio as long as the Jog input is set
```iecst
(********************************************************************
 * COPYRIGHT -- Bernecker + Rainer
 ********************************************************************
 * Library: UserSpilke
 * File: SPR_JogGear.st
 * Author: knausenbergl
 * Created: December 21, 2012
 ********************************************************************
 * Implementation of library UserSpilke
 ********************************************************************)

(*<$Description$> Gear in and update the gear ratio as long as the Jog input is set </$Description$>*)
FUNCTION_BLOCK SPR_JogGear

	IS.R_TRIG_Jog.CLK	:= Jog;
	IS.R_TRIG_Jog();

	IS.MC_ReadStatus_0.Axis := Slave;
	IS.MC_ReadStatus_0.Enable := TRUE;
	IS.MC_ReadStatus_0();

	IS.GearRatioChanged	:=
	(RatioNumerator <> IS.MC_GearIn_0.RatioNumerator)
	OR (RatioDenominator <> IS.MC_GearIn_0.RatioDenominator);

	CASE IS.State OF

		//***************	IDLE	***************
		0:
			IF (IS.R_TRIG_Jog.Q) THEN
				IS.MC_GearIn_0.Acceleration				:= Acceleration;
				IS.MC_GearIn_0.Deceleration				:= Deceleration;
				IS.MC_GearIn_0.MasterParID				:= MasterParID;
				IS.MC_GearIn_0.MasterParIDMaxVelocity	:= MasterParIDMaxVelocity;
				IS.MC_GearIn_0.RatioDenominator			:= RatioDenominator;
				IS.MC_GearIn_0.RatioNumerator			:= RatioNumerator;
				IS.MC_GearIn_0.Execute		:= TRUE;
				IS.State	:= 1;
			END_IF;

		//***************	GEARING IN	***************
		1:
			//error in gear FUB
			IF (IS.MC_GearIn_0.Error) THEN
				Error		:= TRUE;
				ErrorID		:= IS.MC_GearIn_0.ErrorID;
				IS.State	:= 255;
			//gear aborted by FUB other than halt
			ELSIF (IS.MC_GearIn_0.CommandAborted) THEN
				CommandAborted	:= TRUE;
				IS.State		:= 254;
			//trigger halt command
			ELSIF (NOT Jog) THEN
				IS.MC_Halt_0.Deceleration	:= Deceleration;
				IS.State	:= 3;
			//change gear ratio
			ELSIF (IS.GearRatioChanged) THEN
				IS.MC_GearIn_0.Execute	:= FALSE;
				IS.State	:= 100;
			//everything ok
			ELSIF (IS.MC_GearIn_0.InGear) THEN
				IS.State	:= 2;
			END_IF;

		//***************	IN GEAR	***************
		2:
			//error in gear FUB
			IF (IS.MC_GearIn_0.Error) THEN
				Error		:= TRUE;
				ErrorID		:= IS.MC_GearIn_0.ErrorID;
				IS.State	:= 255;
			//gear aborted by FUB other than halt
			ELSIF (IS.MC_GearIn_0.CommandAborted) THEN
				CommandAborted	:= TRUE;
				IS.State	:= 254;
			//trigger halt command
			ELSIF (NOT Jog) THEN
				IS.MC_Halt_0.Deceleration	:= Acceleration;
				IS.State	:= 3;
			//change gear ratio
			ELSIF (IS.GearRatioChanged) THEN
				IS.MC_GearIn_0.Execute	:= FALSE;
				IS.State				:= 100;
			END_IF;

		//***************	TRIGGER HALT	***************
		3:
			//error in gear FUB
			IF (IS.MC_GearIn_0.Error) THEN
				Error		:= TRUE;
				ErrorID		:= IS.MC_GearIn_0.ErrorID;
				IS.State	:= 255;
			//gear aborted by FUB other than halt
			ELSIF (IS.MC_GearIn_0.CommandAborted) THEN
				CommandAborted	:= TRUE;
				IS.State		:= 254;
			//ok to trigger halt command
			ELSE
				IS.MC_GearIn_0.Execute	:= FALSE;
				IF ( IS.MC_ReadStatus_0.DiscreteMotion OR IS.MC_ReadStatus_0.ContinuousMotion OR IS.MC_ReadStatus_0.SynchronizedMotion ) THEN
					IS.MC_Halt_0.Execute	:= TRUE;
				ELSE
				END_IF
				IS.State	:= 254;
			END_IF;

		//***************	HALTING	***************
		4:
			//error in halt FUB
			IF (IS.MC_Halt_0.Error) THEN
				Error		:= TRUE;
				ErrorID		:= IS.MC_Halt_0.ErrorID;
				IS.State	:= 255;
			//halt FUB aborted
			ELSIF (IS.MC_Halt_0.CommandAborted) THEN
				CommandAborted	:= TRUE;
				IS.State		:= 254;
			//everything OK, axis in standstill
			ELSIF (IS.MC_Halt_0.Done) THEN
				IS.State	:= 0;
			END_IF;

		//***************	CHANGE GEAR RATIO	***************
		100:
			IS.MC_GearIn_0.Acceleration				:= Acceleration;
			IS.MC_GearIn_0.Deceleration				:= Deceleration;
			IS.MC_GearIn_0.MasterParID				:= MasterParID;
			IS.MC_GearIn_0.MasterParIDMaxVelocity	:= MasterParIDMaxVelocity;
			IS.MC_GearIn_0.RatioDenominator			:= RatioDenominator;
			IS.MC_GearIn_0.RatioNumerator			:= RatioNumerator;
			IS.MC_GearIn_0.Execute	:= TRUE;
			IS.State	:= 1;

			//error in gear FUB
			IF (IS.MC_GearIn_0.Error) THEN
				Error		:= TRUE;
				ErrorID		:= IS.MC_GearIn_0.ErrorID;
				IS.State	:= 255;
			//gear aborted by FUB other than halt
			ELSIF (IS.MC_GearIn_0.CommandAborted) THEN
				IS.MC_GearIn_0.Execute	:= FALSE;
				CommandAborted			:= TRUE;
				IS.State	:= 254;
			//trigger halt command
			ELSIF (NOT Jog) THEN
				IS.MC_Halt_0.Deceleration	:= Acceleration;
				IS.State	:= 3;
			END_IF;

		//***************	COMMAND ABORTED	***************
		254:
			//FUB reset, go back to init state
			IF (NOT Jog) THEN
				IS.MC_GearIn_0.Execute	:= FALSE;
				IS.MC_Halt_0.Execute	:= FALSE;
				CommandAborted			:= FALSE;
				IS.State	:= 0;
			END_IF;

		//***************	ERROR	***************
		255:
			//FUB reset, go back to init state
			IF (NOT Jog) THEN
				IS.MC_GearIn_0.Execute	:= FALSE;
				IS.MC_Halt_0.Execute	:= FALSE;
				Error		:= FALSE;
				ErrorID		:= ERR_OK;
				IS.State	:= 0;
			END_IF;

	END_CASE

	IS.MC_GearIn_0.Slave	:= Slave;
	IS.MC_GearIn_0.Master	:= Master;
	IS.MC_GearIn_0();

	IS.MC_Halt_0.Axis	:= Slave;
	IS.MC_Halt_0();

	Busy	:= IS.MC_GearIn_0.Busy OR IS.MC_Halt_0.Busy;
	Halting	:= IS.MC_Halt_0.Busy;
	InGear	:= IS.MC_GearIn_0.InGear;

END_FUNCTION_BLOCK
```
